C05457=1086.309,22.215,441.424,174.656,18.933,153.065
C05458=1086.315,22.464,441.409,174.658,18.935,153.065
C05459=1086.320,22.714,441.394,174.659,18.937,153.065
C05460=1086.326,22.963,441.379,174.661,18.939,153.065
C05461=1086.332,23.213,441.365,174.663,18.941,153.066
C05462=1086.337,23.462,441.350,174.664,18.942,153.066
C05463=1086.344,23.712,441.335,174.666,18.944,153.066
C05464=1086.349,23.961,441.320,174.667,18.946,153.066
C05465=1086.354,24.210,441.305,174.669,18.948,153.066
C05466=1086.361,24.460,441.290,174.671,18.951,153.066
C05467=1086.366,24.709,441.276,174.672,18.952,153.066
C05468=1086.372,24.959,441.261,174.674,18.954,153.066
C05469=1086.378,25.208,441.246,174.676,18.956,153.066
C05470=1086.384,25.458,441.231,174.677,18.958,153.066
C05471=1086.389,25.707,441.216,174.680,18.960,153.066
C05472=1086.395,25.957,441.201,174.681,18.962,153.066
C05473=1086.401,26.206,441.187,174.682,18.963,153.067
C05474=1086.407,26.456,441.171,174.684,18.966,153.067
C05475=1086.412,26.705,441.157,174.686,18.967,153.067
C05476=1086.419,26.955,441.142,174.687,18.969,153.067
C05477=1086.424,27.205,441.127,174.689,18.971,153.067
C05478=1086.430,27.454,441.112,174.691,18.973,153.067
C05479=1086.436,27.704,441.097,174.692,18.975,153.067
C05480=1086.442,27.953,441.082,174.694,18.977,153.067
C05481=1086.448,28.203,441.067,174.695,18.979,153.067
C05482=1086.453,28.452,441.052,174.697,18.980,153.067
C05483=1086.459,28.702,441.037,174.699,18.983,153.067
C05484=1086.464,28.951,441.022,174.700,18.984,153.067
C05485=1086.471,29.200,441.007,174.702,18.986,153.068
C05486=1086.476,29.450,440.992,174.704,18.988,153.068
C05487=1086.482,29.699,440.977,174.705,18.990,153.068
C05488=1086.487,29.949,440.962,174.706,18.992,153.068
C05489=1086.494,30.198,440.947,174.709,18.994,153.068
C05490=1086.499,30.448,440.931,174.710,18.996,153.068
C05491=1086.505,30.697,440.916,174.711,18.997,153.068
C05492=1086.512,30.975,440.899,174.713,19.000,153.068
C05493=1086.518,31.253,440.883,174.716,19.002,153.068
C05494=1086.524,31.531,440.866,174.717,19.004,153.068
C05495=1086.530,31.809,440.848,174.719,19.006,153.068
C05496=1086.536,32.058,440.833,174.720,19.008,153.069
C05497=1086.542,32.308,440.818,174.723,19.010,153.069
C05498=1086.548,32.557,440.803,174.724,19.012,153.069
C05499=1086.554,32.807,440.788,174.725,19.014,153.069
C05500=1086.559,33.056,440.773,174.728,19.016,153.069
C05501=1086.565,33.306,440.758,174.729,19.017,153.069
C05502=1086.571,33.555,440.743,174.731,19.020,153.069
C05503=1086.576,33.805,440.728,174.732,19.021,153.069
C05504=1086.582,34.055,440.712,174.734,19.023,153.069
C05505=1086.588,34.303,440.697,174.736,19.025,153.069
C05506=1086.594,34.553,440.681,174.737,19.027,153.069
C05507=1086.600,34.802,440.667,174.739,19.029,153.069
C05508=1086.605,35.052,440.651,174.741,19.031,153.069
C05509=1086.612,35.302,440.636,174.742,19.033,153.070
C05510=1086.617,35.551,440.620,174.745,19.035,153.070
C05511=1086.623,35.801,440.605,174.746,19.037,153.070
C05512=1086.629,36.050,440.590,174.747,19.038,153.070
C05513=1086.634,36.299,440.575,174.750,19.040,153.070
C05514=1086.640,36.549,440.560,174.751,19.042,153.070
C05515=1086.646,36.798,440.544,174.752,19.044,153.070
C05516=1086.651,37.048,440.528,174.754,19.046,153.070
C05517=1086.658,37.297,440.513,174.756,19.047,153.070
C05518=1086.663,37.547,440.498,174.758,19.050,153.070
C05519=1086.669,37.796,440.482,174.759,19.051,153.070
C05520=1086.675,38.046,440.467,174.761,19.053,153.070
C05521=1086.680,38.295,440.452,174.763,19.056,153.070
C05522=1086.686,38.545,440.436,174.764,19.057,153.070
C05523=1086.692,38.794,440.420,174.766,19.059,153.071
C05524=1086.698,39.043,440.405,174.768,19.061,153.071
C05525=1086.703,39.293,440.390,174.769,19.063,153.071
C05526=1086.709,39.543,440.373,174.772,19.065,153.071
C05527=1086.714,39.792,440.358,174.773,19.067,153.071
C05528=1086.721,40.041,440.343,174.774,19.068,153.071
C05529=1086.727,40.291,440.327,174.776,19.070,153.071
C05530=1086.732,40.540,440.312,174.778,19.072,153.071
C05531=1086.737,40.790,440.296,174.780,19.074,153.071
C05532=1086.744,41.039,440.281,174.781,19.076,153.071
C05533=1086.749,41.288,440.266,174.783,19.078,153.071
C05534=1086.755,41.538,440.250,174.785,19.080,153.071
C05535=1086.761,41.788,440.234,174.786,19.081,153.071
C05536=1086.766,42.037,440.219,174.788,19.084,153.072
C05537=1086.772,42.286,440.203,174.790,19.086,153.072
C05538=1086.778,42.536,440.187,174.791,19.087,153.072
C05539=1086.783,42.785,440.172,174.793,19.090,153.072
C05540=1086.789,43.035,440.156,174.795,19.091,153.072
C05541=1086.795,43.285,440.140,174.796,19.093,153.072
C05542=1086.801,43.534,440.124,174.798,19.095,153.072
C05543=1086.806,43.783,440.110,174.800,19.097,153.072
C05544=1086.812,44.032,440.093,174.802,19.099,153.072
C05545=1086.818,44.282,440.078,174.803,19.100,153.072
C05546=1086.823,44.531,440.062,174.805,19.102,153.072
C05547=1086.829,44.781,440.046,174.807,19.104,153.072
C05548=1086.835,45.030,440.030,174.808,19.106,153.072
C05549=1086.840,45.279,440.015,174.810,19.108,153.073
C05550=1086.846,45.529,439.999,174.812,19.110,153.073
C05551=1086.852,45.779,439.983,174.814,19.112,153.073
C05552=1086.857,46.027,439.967,174.815,19.114,153.073
C05553=1086.863,46.277,439.952,174.817,19.116,153.073
C05554=1086.868,46.527,439.935,174.819,19.118,153.073
C05555=1086.874,46.777,439.920,174.820,19.120,153.073
C05556=1086.880,47.055,439.902,174.822,19.122,153.073
C05557=1086.886,47.333,439.884,174.825,19.124,153.073
C05558=1086.893,47.610,439.867,174.826,19.126,153.073
C05559=1086.899,47.888,439.849,174.828,19.128,153.073
C05560=1086.904,48.138,439.833,174.829,19.130,153.073
C05561=1086.910,48.387,439.817,174.832,19.132,153.073
C05562=1086.916,48.636,439.801,174.833,19.134,153.074
C05563=1086.921,48.886,439.786,174.835,19.136,153.074
C05564=1086.927,49.135,439.769,174.837,19.137,153.074
C05565=1086.932,49.385,439.754,174.838,19.139,153.074
C05566=1086.938,49.634,439.738,174.840,19.141,153.074
C05567=1086.944,49.883,439.722,174.842,19.143,153.074
C05568=1086.950,50.133,439.706,174.844,19.145,153.074
C05569=1086.956,50.383,439.690,174.845,19.147,153.074
C05570=1086.961,50.631,439.674,174.847,19.149,153.074
C05571=1086.967,50.881,439.658,174.849,19.151,153.074
C05572=1086.972,51.131,439.642,174.850,19.152,153.074
C05573=1086.978,51.380,439.625,174.853,19.154,153.074
C05574=1086.984,51.630,439.610,174.854,19.156,153.074
C05575=1086.989,51.879,439.594,174.856,19.158,153.074
C05576=1086.995,52.128,439.578,174.857,19.160,153.074
C05577=1087.001,52.378,439.561,174.860,19.162,153.074
C05578=1087.007,52.628,439.546,174.861,19.164,153.075
C05579=1087.013,52.877,439.530,174.862,19.165,153.075
C05580=1087.018,53.126,439.514,174.865,19.167,153.075
C05581=1087.024,53.375,439.497,174.866,19.169,153.075
C05582=1087.029,53.625,439.482,174.868,19.171,153.075
C05583=1087.035,53.875,439.465,174.870,19.173,153.075
C05584=1087.041,54.124,439.449,174.872,19.175,153.075
C05585=1087.047,54.373,439.432,174.873,19.176,153.075
C05586=1087.053,54.623,439.416,174.875,19.178,153.075
C05587=1087.058,54.872,439.401,174.877,19.180,153.075
C05588=1087.064,55.121,439.385,174.878,19.182,153.075
C05589=1087.069,55.371,439.369,174.881,19.184,153.075
C05590=1087.075,55.620,439.352,174.882,19.186,153.075
C05591=1087.081,55.870,439.335,174.884,19.188,153.075
C05592=1087.087,56.119,439.319,174.886,19.189,153.075
C05593=1087.092,56.369,439.304,174.887,19.191,153.075
C05594=1087.098,56.618,439.287,174.890,19.193,153.075
C05595=1087.104,56.868,439.271,174.891,19.195,153.076
C05596=1087.110,57.117,439.255,174.893,19.197,153.076
C05597=1087.115,57.366,439.239,174.894,19.198,153.076
C05598=1087.121,57.615,439.222,174.897,19.200,153.076
C05599=1087.127,57.865,439.206,174.898,19.202,153.076
C05600=1087.133,58.114,439.190,174.901,19.204,153.076
C05601=1087.139,58.363,439.173,174.902,19.205,153.076
C05602=1087.144,58.613,439.157,174.903,19.207,153.076
C05603=1087.150,58.862,439.141,174.905,19.209,153.076
C05604=1087.155,59.112,439.125,174.907,19.211,153.076
C05605=1087.161,59.362,439.108,174.909,19.213,153.076
C05606=1087.167,59.611,439.092,174.911,19.215,153.076
C05607=1087.173,59.860,439.076,174.913,19.217,153.076
C05608=1087.179,60.110,439.060,174.914,19.218,153.076
C05609=1087.184,60.359,439.043,174.917,19.220,153.076
C05610=1087.190,60.609,439.027,174.918,19.222,153.076
C05611=1087.196,60.858,439.010,174.920,19.224,153.076
C05612=1087.202,61.107,438.994,174.922,19.225,153.076
C05613=1087.208,61.357,438.978,174.923,19.227,153.076
C05614=1087.214,61.606,438.960,174.926,19.229,153.076
C05615=1087.220,61.855,438.944,174.927,19.230,153.076
C05616=1087.226,62.104,438.928,174.929,19.233,153.076
C05617=1087.232,62.354,438.911,174.931,19.234,153.076
C05618=1087.237,62.603,438.895,174.933,19.236,153.076
C05619=1087.243,62.853,438.878,174.934,19.238,153.076
C05620=1087.249,63.130,438.860,174.937,19.240,153.076
C05621=1087.256,63.408,438.842,174.939,19.242,153.076
C05622=1087.262,63.686,438.824,174.940,19.243,153.077
C05623=1087.269,63.964,438.805,174.943,19.245,153.077
C05624=1087.275,64.213,438.789,174.945,19.247,153.077
C05625=1087.280,64.462,438.772,174.946,19.249,153.077
C05626=1087.286,64.712,438.755,174.948,19.251,153.077
C05627=1087.292,64.961,438.739,174.950,19.253,153.077
C05628=1087.297,65.211,438.722,174.952,19.254,153.077
C05629=1087.303,65.460,438.706,174.954,19.256,153.077
C05630=1087.308,65.710,438.689,174.955,19.258,153.077
C05631=1087.315,65.958,438.672,174.957,19.260,153.077
C05632=1087.320,66.208,438.655,174.959,19.262,153.077
C05633=1087.326,66.457,438.639,174.961,19.264,153.077
C05634=1087.332,66.707,438.623,174.963,19.265,153.077
C05635=1087.337,66.956,438.606,174.965,19.267,153.077
C05636=1087.344,67.206,438.589,174.966,19.269,153.077
C05637=1087.349,67.455,438.572,174.969,19.271,153.077
C05638=1087.355,67.705,438.556,174.970,19.272,153.077
C05639=1087.360,67.954,438.539,174.972,19.274,153.077
C05640=1087.366,68.203,438.522,174.974,19.276,153.077
C05641=1087.372,68.453,438.505,174.976,19.278,153.077
C05642=1087.378,68.702,438.489,174.978,19.279,153.077
C05643=1087.383,68.952,438.472,174.980,19.281,153.077
C05644=1087.389,69.201,438.455,174.981,19.283,153.077
C05645=1087.394,69.450,438.438,174.984,19.285,153.077
C05646=1087.400,69.700,438.422,174.985,19.286,153.077
C05647=1087.406,69.949,438.404,174.987,19.288,153.077
C05648=1087.412,70.198,438.388,174.989,19.290,153.077
C05649=1087.417,70.448,438.371,174.990,19.292,153.077
C05650=1087.422,70.697,438.353,174.992,19.294,153.077
C05651=1087.428,70.946,438.337,174.994,19.295,153.077
C05652=1087.434,71.196,438.320,174.996,19.297,153.077
C05653=1087.440,71.445,438.303,174.998,19.299,153.078
C05654=1087.446,71.695,438.286,175.000,19.301,153.078
C05655=1087.451,71.944,438.269,175.001,19.302,153.078
C05656=1087.457,72.193,438.252,175.004,19.304,153.078
C05657=1087.462,72.443,438.235,175.005,19.306,153.078
C05658=1087.469,72.691,438.218,175.007,19.308,153.078
C05659=1087.474,72.941,438.202,175.009,19.309,153.078
C05660=1087.479,73.191,438.185,175.011,19.311,153.078
C05661=1087.485,73.440,438.168,175.013,19.313,153.078
C05662=1087.490,73.689,438.151,175.015,19.315,153.078
C05663=1087.497,73.939,438.133,175.016,19.316,153.078
C05664=1087.503,74.188,438.117,175.019,19.318,153.078
C05665=1087.508,74.437,438.099,175.020,19.320,153.078
C05666=1087.513,74.687,438.082,175.022,19.322,153.078
C05667=1087.520,74.936,438.065,175.024,19.323,153.078
C05668=1087.525,75.185,438.049,175.026,19.325,153.078
C05669=1087.530,75.434,438.031,175.028,19.327,153.078
C05670=1087.537,75.684,438.014,175.030,19.329,153.078
C05671=1087.542,75.934,437.997,175.031,19.330,153.078
C05672=1087.548,76.183,437.980,175.034,19.332,153.078
C05673=1087.554,76.432,437.963,175.035,19.334,153.078
C05674=1087.559,76.682,437.946,175.038,19.336,153.078
C05675=1087.565,76.931,437.929,175.039,19.337,153.078
C05676=1087.571,77.180,437.911,175.041,19.339,153.078
C05677=1087.577,77.430,437.894,175.043,19.341,153.078
C05678=1087.582,77.679,437.877,175.045,19.343,153.078
C05679=1087.587,77.928,437.860,175.047,19.344,153.078
C05680=1087.593,78.177,437.842,175.049,19.346,153.078
C05681=1087.599,78.427,437.826,175.051,19.348,153.078
C05682=1087.605,78.677,437.808,175.053,19.350,153.078
C05683=1087.610,78.926,437.791,175.055,19.352,153.078
C05684=1087.617,79.203,437.772,175.056,19.353,153.078
C05685=1087.623,79.481,437.752,175.059,19.355,153.078
C05686=1087.629,79.758,437.734,175.061,19.357,153.078
C05687=1087.636,80.036,437.713,175.063,19.359,153.078
C05688=1087.641,80.286,437.697,175.065,19.361,153.078
C05689=1087.646,80.535,437.679,175.067,19.363,153.078
C05690=1087.652,80.784,437.661,175.069,19.364,153.078
C05691=1087.657,81.034,437.645,175.071,19.366,153.078
C05692=1087.664,81.283,437.627,175.073,19.367,153.078
C05693=1087.669,81.532,437.610,175.075,19.369,153.078
C05694=1087.675,81.782,437.593,175.076,19.371,153.078
C05695=1087.680,82.031,437.575,175.079,19.373,153.078
C05696=1087.689,82.421,437.547,175.082,19.375,153.078
C05697=1087.698,82.811,437.520,175.085,19.378,153.078
C05698=1087.707,83.200,437.494,175.088,19.381,153.078
C05699=1087.716,83.590,437.466,175.091,19.384,153.078
C05700=1087.721,83.839,437.449,175.092,19.385,153.078
C05701=1087.727,84.089,437.431,175.095,19.387,153.078
C05702=1087.733,84.338,437.413,175.096,19.389,153.078
C05703=1087.738,84.587,437.396,175.098,19.391,153.078
C05704=1087.744,84.836,437.378,175.100,19.392,153.078
C05705=1087.750,85.086,437.360,175.102,19.394,153.078
C05706=1087.755,85.336,437.344,175.105,19.396,153.078
C05707=1087.761,85.585,437.326,175.106,19.397,153.078
C05708=1087.767,85.835,437.308,175.108,19.399,153.078
C05709=1087.772,86.084,437.290,175.110,19.401,153.078
C05710=1087.778,86.333,437.273,175.112,19.402,153.078
C05711=1087.783,86.582,437.255,175.114,19.404,153.078
C05712=1087.789,86.831,437.237,175.116,19.406,153.078
C05713=1087.795,87.080,437.220,175.118,19.407,153.078
C05714=1087.800,87.329,437.202,175.120,19.409,153.078
C05715=1087.806,87.580,437.185,175.122,19.410,153.078
C05716=1087.812,87.829,437.168,175.124,19.412,153.078
C05717=1087.817,88.078,437.150,175.126,19.414,153.078
C05718=1087.823,88.328,437.132,175.128,19.415,153.078
C05719=1087.829,88.577,437.114,175.130,19.417,153.078
C05720=1087.834,88.826,437.097,175.132,19.419,153.078
C05721=1087.840,89.075,437.079,175.134,19.421,153.078
C05722=1087.846,89.325,437.061,175.136,19.422,153.078
C05723=1087.852,89.574,437.043,175.138,19.424,153.078
C05724=1087.858,89.823,437.026,175.139,19.425,153.078
C05725=1087.863,90.072,437.008,175.142,19.427,153.078
C05726=1087.869,90.322,436.990,175.144,19.429,153.078
C05727=1087.875,90.571,436.973,175.146,19.430,153.078
C05728=1087.880,90.820,436.955,175.148,19.432,153.078
C05729=1087.886,91.070,436.937,175.150,19.434,153.078
C05730=1087.892,91.319,436.920,175.152,19.436,153.078
C05731=1087.897,91.568,436.902,175.153,19.437,153.078
C05732=1087.903,91.817,436.883,175.156,19.439,153.078
C05733=1087.909,92.066,436.865,175.157,19.440,153.078
C05734=1087.915,92.316,436.847,175.160,19.442,153.078
C05735=1087.920,92.565,436.830,175.162,19.444,153.078
C05736=1087.925,92.815,436.812,175.164,19.445,153.078
C05737=1087.931,93.064,436.794,175.166,19.447,153.078
C05738=1087.937,93.313,436.776,175.168,19.449,153.078
C05739=1087.942,93.562,436.759,175.170,19.451,153.078
C05740=1087.948,93.812,436.741,175.172,19.452,153.078
C05741=1087.953,94.061,436.722,175.174,19.454,153.078
C05742=1087.959,94.310,436.704,175.176,19.456,153.078
C05743=1087.965,94.560,436.686,175.178,19.457,153.078
C05744=1087.974,94.947,436.658,175.181,19.459,153.078
C05745=1087.982,95.333,436.630,175.184,19.462,153.078
C05746=1087.991,95.720,436.602,175.187,19.465,153.078
C05747=1088.000,96.106,436.575,175.190,19.467,153.078
C05748=1088.006,96.355,436.556,175.193,19.469,153.078
C05749=1088.011,96.604,436.538,175.194,19.470,153.078
C05750=1088.017,96.854,436.520,175.197,19.472,153.078
C05751=1088.022,97.103,436.503,175.198,19.473,153.078
C05752=1088.028,97.353,436.483,175.200,19.475,153.078
C05753=1088.034,97.602,436.466,175.203,19.477,153.078
C05754=1088.040,97.851,436.448,175.204,19.478,153.078
C05755=1088.046,98.100,436.430,175.207,19.480,153.078
C05756=1088.051,98.350,436.411,175.208,19.481,153.078
C05757=1088.056,98.599,436.394,175.211,19.483,153.078
C05758=1088.063,98.849,436.376,175.213,19.485,153.078
C05759=1088.068,99.097,436.357,175.215,19.486,153.078
C05760=1088.073,99.346,436.339,175.217,19.488,153.077
C05761=1088.079,99.596,436.321,175.219,19.490,153.078
C05762=1088.085,99.846,436.302,175.221,19.492,153.078
C05763=1088.090,100.095,436.284,175.224,19.493,153.077
C05764=1088.097,100.344,436.266,175.225,19.495,153.077
C05765=1088.102,100.593,436.248,175.228,19.496,153.077
C05766=1088.108,100.843,436.230,175.229,19.498,153.077
C05767=1088.114,101.091,436.211,175.232,19.499,153.077
C05768=1088.119,101.341,436.193,175.234,19.501,153.077
C05769=1088.125,101.590,436.175,175.236,19.502,153.077
C05770=1088.130,101.840,436.156,175.238,19.504,153.077
C05771=1088.136,102.088,436.138,175.239,19.506,153.077
C05772=1088.141,102.338,436.119,175.242,19.507,153.077
C05773=1088.147,102.587,436.102,175.244,19.509,153.077
C05774=1088.153,102.837,436.082,175.246,19.510,153.077
C05775=1088.158,103.086,436.065,175.248,19.512,153.077
C05776=1088.164,103.335,436.046,175.250,19.513,153.077
C05777=1088.169,103.584,436.028,175.252,19.515,153.077
C05778=1088.175,103.834,436.009,175.255,19.517,153.077
C05779=1088.181,104.083,435.991,175.256,19.518,153.077
C05780=1088.186,104.332,435.972,175.259,19.520,153.077
C05781=1088.192,104.581,435.954,175.260,19.521,153.077
C05782=1088.197,104.831,435.935,175.263,19.523,153.077
C05783=1088.203,105.079,435.917,175.265,19.525,153.077
C05784=1088.209,105.329,435.898,175.267,19.526,153.077
C05785=1088.214,105.578,435.880,175.269,19.528,153.077
C05786=1088.220,105.828,435.862,175.271,19.530,153.077
C05787=1088.226,106.077,435.842,175.273,19.531,153.077
C05788=1088.231,106.326,435.825,175.275,19.533,153.077
C05789=1088.237,106.575,435.806,175.277,19.534,153.076
C05790=1088.243,106.824,435.787,175.279,19.536,153.076
C05791=1088.248,107.074,435.769,175.282,19.537,153.076
C05792=1088.253,107.323,435.750,175.283,19.539,153.076
C05793=1088.259,107.572,435.731,175.286,19.540,153.076
C05794=1088.265,107.822,435.713,175.287,19.542,153.076
C05795=1088.271,108.070,435.694,175.290,19.543,153.076
C05796=1088.276,108.320,435.676,175.292,19.545,153.076
C05797=1088.282,108.570,435.657,175.294,19.546,153.076
C05798=1088.288,108.818,435.638,175.296,19.548,153.076
C05799=1088.293,109.068,435.619,175.299,19.550,153.076
C05800=1088.299,109.317,435.602,175.300,19.551,153.076
C05801=1088.304,109.566,435.582,175.303,19.553,153.076
C05802=1088.310,109.816,435.563,175.305,19.555,153.076
C05803=1088.316,110.065,435.545,175.307,19.556,153.076
C05804=1088.321,110.314,435.526,175.309,19.558,153.076
C05805=1088.328,110.563,435.508,175.311,19.559,153.076
C05806=1088.333,110.812,435.489,175.314,19.560,153.075
C05807=1088.338,111.062,435.470,175.316,19.562,153.075
C05808=1088.345,111.339,435.449,175.318,19.564,153.075
C05809=1088.351,111.617,435.428,175.321,19.566,153.075
C05810=1088.358,111.895,435.407,175.323,19.567,153.075
C05811=1088.364,112.173,435.386,175.325,19.568,153.075
C05812=1088.369,112.422,435.367,175.327,19.570,153.075
C05813=1088.375,112.671,435.348,175.330,19.572,153.075
C05814=1088.381,112.921,435.330,175.331,19.573,153.075
C05815=1088.386,113.170,435.311,175.334,19.575,153.075
C05816=1088.392,113.419,435.292,175.336,19.576,153.075
C05817=1088.398,113.668,435.273,175.338,19.578,153.075
C05818=1088.403,113.917,435.254,175.340,19.579,153.075
C05819=1088.409,114.166,435.235,175.343,19.581,153.075
C05820=1088.414,114.416,435.216,175.344,19.582,153.075
C05821=1088.420,114.664,435.197,175.347,19.584,153.075
C05822=1088.426,114.914,435.179,175.349,19.586,153.075
C05823=1088.431,115.164,435.160,175.351,19.587,153.074
C05824=1088.436,115.412,435.141,175.353,19.588,153.074
C05825=1088.442,115.662,435.122,175.356,19.590,153.074
C05826=1088.448,115.911,435.102,175.357,19.591,153.074
C05827=1088.453,116.160,435.083,175.360,19.593,153.074
C05828=1088.459,116.409,435.064,175.362,19.595,153.074
C05829=1088.464,116.659,435.045,175.364,19.596,153.074
C05830=1088.469,116.908,435.026,175.366,19.598,153.074
C05831=1088.475,117.157,435.007,175.369,19.599,153.074
C05832=1088.481,117.406,434.988,175.371,19.600,153.074
C05833=1088.486,117.656,434.968,175.373,19.602,153.074
C05834=1088.491,117.905,434.949,175.375,19.604,153.074
C05835=1088.497,118.154,434.930,175.377,19.605,153.074
C05836=1088.503,118.403,434.911,175.379,19.607,153.074
C05837=1088.508,118.652,434.892,175.382,19.608,153.074
C05838=1088.514,118.902,434.873,175.384,19.609,153.073
C05839=1088.519,119.151,434.854,175.386,19.611,153.073
C05840=1088.525,119.400,434.834,175.388,19.613,153.073
C05841=1088.530,119.649,434.815,175.390,19.614,153.073
C05842=1088.536,119.898,434.796,175.392,19.616,153.073
C05843=1088.542,120.147,434.776,175.395,19.617,153.073
C05844=1088.547,120.397,434.757,175.397,19.618,153.073
C05845=1088.553,120.646,434.738,175.399,19.620,153.073
C05846=1088.558,120.895,434.719,175.402,19.622,153.073
C05847=1088.564,121.144,434.700,175.403,19.623,153.073
C05848=1088.570,121.394,434.680,175.406,19.625,153.073
C05849=1088.575,121.643,434.661,175.408,19.627,153.073
C05850=1088.581,121.891,434.642,175.410,19.628,153.073
C05851=1088.586,122.141,434.622,175.412,19.629,153.073
C05852=1088.592,122.390,434.603,175.415,19.631,153.072
C05853=1088.598,122.640,434.584,175.417,19.632,153.072
C05854=1088.603,122.889,434.565,175.419,19.634,153.072
C05855=1088.609,123.137,434.545,175.421,19.635,153.072
C05856=1088.615,123.387,434.526,175.424,19.637,153.072
C05857=1088.620,123.636,434.507,175.426,19.638,153.072
C05858=1088.626,123.886,434.487,175.428,19.639,153.072
C05859=1088.632,124.134,434.467,175.431,19.641,153.072
C05860=1088.638,124.384,434.448,175.432,19.642,153.072
C05861=1088.643,124.633,434.429,175.435,19.644,153.072
C05862=1088.648,124.882,434.410,175.437,19.645,153.072
C05863=1088.654,125.131,434.389,175.439,19.646,153.071
C05864=1088.659,125.381,434.370,175.442,19.648,153.071
C05865=1088.665,125.630,434.351,175.444,19.649,153.071
C05866=1088.671,125.879,434.331,175.446,19.651,153.071
C05867=1088.677,126.128,434.312,175.448,19.652,153.071
C05868=1088.682,126.378,434.292,175.451,19.654,153.071
C05869=1088.688,126.626,434.273,175.453,19.655,153.071
C05870=1088.693,126.875,434.254,175.455,19.656,153.071
C05871=1088.699,127.125,434.234,175.457,19.658,153.071
C05872=1088.706,127.402,434.212,175.460,19.659,153.071
C05873=1088.712,127.680,434.190,175.463,19.661,153.070
C05874=1088.718,127.958,434.169,175.465,19.662,153.070
C05875=1088.725,128.235,434.146,175.468,19.664,153.070
C05876=1088.730,128.485,434.127,175.470,19.666,153.070
C05877=1088.735,128.734,434.107,175.473,19.667,153.070
C05878=1088.741,128.983,434.087,175.474,19.668,153.070
C05879=1088.747,129.233,434.068,175.477,19.670,153.070
C05880=1088.753,129.481,434.048,175.479,19.671,153.070
C05881=1088.759,129.731,434.029,175.481,19.672,153.070
C05882=1088.765,129.980,434.009,175.484,19.674,153.069
C05883=1088.770,130.229,433.990,175.486,19.675,153.069
C05884=1088.776,130.478,433.969,175.489,19.677,153.069
C05885=1088.781,130.728,433.950,175.490,19.678,153.069
C05886=1088.787,130.976,433.930,175.493,19.679,153.069
C05887=1088.793,131.226,433.911,175.495,19.681,153.069
C05888=1088.799,131.475,433.891,175.498,19.682,153.069
C05889=1088.804,131.724,433.871,175.500,19.683,153.069
C05890=1088.810,131.973,433.851,175.502,19.685,153.069
C05891=1088.816,132.222,433.831,175.505,19.686,153.068
C05892=1088.822,132.471,433.812,175.506,19.687,153.068
C05893=1088.827,132.721,433.791,175.509,19.689,153.068
C05894=1088.833,132.970,433.772,175.512,19.691,153.068
C05895=1088.839,133.219,433.752,175.514,19.692,153.068
C05896=1088.844,133.468,433.732,175.516,19.693,153.068
C05897=1088.850,133.717,433.712,175.518,19.695,153.068
C05898=1088.855,133.967,433.692,175.521,19.696,153.068
C05899=1088.860,134.215,433.673,175.523,19.698,153.067
C05900=1088.866,134.464,433.653,175.525,19.699,153.067
C05901=1088.871,134.713,433.632,175.528,19.700,153.067
C05902=1088.877,134.963,433.613,175.530,19.702,153.067
C05903=1088.882,135.212,433.593,175.533,19.703,153.067
C05904=1088.888,135.461,433.573,175.534,19.704,153.067
C05905=1088.894,135.710,433.553,175.537,19.706,153.067
C05906=1088.900,135.960,433.532,175.540,19.707,153.067
C05907=1088.906,136.209,433.512,175.542,19.709,153.067
C05908=1088.911,136.458,433.492,175.544,19.710,153.066
C05909=1088.917,136.707,433.473,175.546,19.711,153.066
C05910=1088.923,136.956,433.453,175.549,19.713,153.066
C05911=1088.928,137.205,433.432,175.551,19.714,153.066
C05912=1088.934,137.454,433.412,175.553,19.715,153.066
C05913=1088.939,137.704,433.392,175.556,19.716,153.066
C05914=1088.945,137.953,433.372,175.558,19.718,153.066
C05915=1088.950,138.202,433.352,175.561,19.719,153.066
C05916=1088.956,138.450,433.332,175.563,19.720,153.065
C05917=1088.961,138.700,433.311,175.565,19.722,153.065
C05918=1088.967,138.949,433.292,175.568,19.723,153.065
C05919=1088.972,139.198,433.272,175.570,19.725,153.065
C05920=1088.978,139.447,433.252,175.572,19.726,153.065
C05921=1088.983,139.696,433.231,175.575,19.727,153.065
C05922=1088.989,139.945,433.211,175.577,19.729,153.065
C05923=1088.995,140.195,433.190,175.580,19.730,153.065
C05924=1089.001,140.444,433.170,175.582,19.731,153.064
C05925=1089.007,140.693,433.150,175.584,19.732,153.064
C05926=1089.012,140.942,433.130,175.587,19.734,153.064
C05927=1089.018,141.191,433.110,175.589,19.735,153.064
C05928=1089.023,141.440,433.089,175.592,19.737,153.064
C05929=1089.029,141.689,433.069,175.594,19.738,153.064
C05930=1089.034,141.938,433.049,175.596,19.739,153.064
C05931=1089.039,142.187,433.028,175.599,19.741,153.064
C05932=1089.045,142.436,433.008,175.601,19.742,153.063
C05933=1089.051,142.685,432.988,175.604,19.744,153.063
C05934=1089.056,142.935,432.967,175.606,19.744,153.063
C05935=1089.062,143.184,432.947,175.608,19.746,153.063
C05936=1089.068,143.461,432.924,175.611,19.747,153.063
C05937=1089.075,143.739,432.902,175.613,19.749,153.063
C05938=1089.081,144.017,432.878,175.616,19.750,153.063
C05939=1089.086,144.294,432.856,175.619,19.753,153.062
C05940=1089.093,144.544,432.835,175.621,19.753,153.062
C05941=1089.098,144.793,432.815,175.624,19.755,153.062
C05942=1089.104,145.042,432.794,175.626,19.756,153.062
C05943=1089.109,145.291,432.774,175.629,19.758,153.062
C05944=1089.115,145.540,432.754,175.631,19.759,153.062
C05945=1089.120,145.789,432.733,175.633,19.760,153.061
C05946=1089.126,146.039,432.712,175.636,19.761,153.061
C05947=1089.132,146.287,432.692,175.638,19.763,153.061
C05948=1089.137,146.536,432.671,175.641,19.764,153.061
C05949=1089.143,146.785,432.650,175.643,19.766,153.061
C05950=1089.149,147.034,432.630,175.645,19.766,153.061
C05951=1089.155,147.284,432.610,175.648,19.768,153.061
C05952=1089.160,147.533,432.589,175.650,19.769,153.061
C05953=1089.165,147.781,432.568,175.653,19.770,153.060
C05954=1089.171,148.030,432.548,175.656,19.772,153.060
C05955=1089.177,148.280,432.527,175.658,19.773,153.060
C05956=1089.182,148.529,432.506,175.660,19.774,153.060
C05957=1089.188,148.778,432.486,175.663,19.776,153.060
C05958=1089.194,149.027,432.465,175.665,19.777,153.060
C05959=1089.199,149.276,432.445,175.668,19.778,153.059
C05960=1089.205,149.526,432.424,175.670,19.779,153.059
C05961=1089.210,149.775,432.403,175.672,19.781,153.059
C05962=1089.216,150.023,432.382,175.675,19.782,153.059
C05963=1089.221,150.272,432.361,175.678,19.783,153.059
C05964=1089.227,150.522,432.340,175.680,19.785,153.059
C05965=1089.232,150.771,432.320,175.683,19.786,153.058
C05966=1089.239,151.019,432.299,175.685,19.787,153.058
C05967=1089.244,151.269,432.279,175.687,19.788,153.058
C05968=1089.249,151.518,432.258,175.690,19.790,153.058
C05969=1089.255,151.767,432.236,175.692,19.791,153.058
C05970=1089.261,152.016,432.216,175.695,19.792,153.058
C05971=1089.266,152.265,432.195,175.698,19.794,153.058
C05972=1089.272,152.514,432.174,175.699,19.795,153.058
C05973=1089.277,152.763,432.153,175.702,19.796,153.057
C05974=1089.283,153.012,432.132,175.705,19.797,153.057
C05975=1089.288,153.261,432.111,175.707,19.799,153.057
C05976=1089.294,153.511,432.090,175.710,19.800,153.057
C05977=1089.299,153.759,432.069,175.712,19.801,153.057
C05978=1089.305,154.009,432.048,175.714,19.803,153.057
C05979=1089.311,154.258,432.027,175.717,19.804,153.056
C05980=1089.316,154.507,432.006,175.719,19.805,153.056
C05981=1089.322,154.755,431.985,175.722,19.807,153.056
C05982=1089.328,155.005,431.965,175.725,19.808,153.056
C05983=1089.334,155.254,431.944,175.727,19.809,153.056
C05984=1089.339,155.502,431.923,175.729,19.810,153.055
C05985=1089.345,155.752,431.902,175.732,19.811,153.055
C05986=1089.350,156.001,431.880,175.734,19.813,153.055
C05987=1089.355,156.250,431.860,175.737,19.814,153.055
C05988=1089.361,156.499,431.838,175.740,19.815,153.055
C05989=1089.367,156.748,431.817,175.742,19.817,153.055
C05990=1089.372,156.997,431.796,175.745,19.818,153.054
C05991=1089.378,157.246,431.775,175.747,19.819,153.054
C05992=1089.383,157.495,431.754,175.749,19.820,153.054
C05993=1089.389,157.744,431.733,175.752,19.821,153.054
C05994=1089.395,157.994,431.712,175.755,19.823,153.054
C05995=1089.400,158.242,431.690,175.757,19.824,153.054
C05996=1089.406,158.491,431.669,175.760,19.825,153.053
C05997=1089.412,158.741,431.648,175.762,19.827,153.053
C05998=1089.417,158.989,431.626,175.765,19.828,153.053
C05999=1089.422,159.239,431.606,175.767,19.829,153.053
C06000=1089.428,159.516,431.582,175.771,19.830,153.053
C06001=1089.435,159.793,431.558,175.773,19.832,153.053
C06002=1089.441,160.071,431.534,175.776,19.833,153.052
C06003=1089.448,160.348,431.510,175.778,19.834,153.052
C06004=1089.453,160.597,431.490,175.781,19.835,153.052
C06005=1089.459,160.846,431.468,175.784,19.837,153.052
C06006=1089.465,161.095,431.447,175.787,19.838,153.052
C06007=1089.470,161.344,431.425,175.789,19.839,153.051
C06008=1089.475,161.593,431.404,175.792,19.840,153.051
C06009=1089.481,161.842,431.383,175.794,19.841,153.051
C06010=1089.487,162.091,431.361,175.796,19.843,153.051
C06011=1089.492,162.341,431.340,175.799,19.844,153.051
C06012=1089.497,162.589,431.319,175.801,19.846,153.051
C06013=1089.503,162.839,431.297,175.804,19.847,153.050
C06014=1089.508,163.087,431.275,175.807,19.848,153.050
C06015=1089.514,163.336,431.254,175.809,19.850,153.050
C06016=1089.519,163.586,431.233,175.812,19.851,153.050
C06017=1089.524,163.834,431.211,175.815,19.852,153.050
C06018=1089.530,164.084,431.189,175.817,19.854,153.050
C06019=1089.535,164.332,431.168,175.819,19.854,153.049
C06020=1089.541,164.581,431.146,175.822,19.856,153.049
C06021=1089.546,164.830,431.124,175.824,19.857,153.049
C06022=1089.552,165.079,431.103,175.827,19.858,153.049
C06023=1089.557,165.329,431.082,175.830,19.860,153.049
C06024=1089.563,165.577,431.060,175.832,19.861,153.049
C06025=1089.568,165.827,431.038,175.835,19.862,153.048
C06026=1089.574,166.075,431.017,175.837,19.864,153.048
C06027=1089.579,166.325,430.995,175.840,19.865,153.048
C06028=1089.585,166.573,430.973,175.843,19.866,153.048
C06029=1089.590,166.822,430.952,175.846,19.867,153.048
C06030=1089.595,167.071,430.930,175.847,19.868,153.048
C06031=1089.601,167.320,430.909,175.850,19.869,153.047
C06032=1089.606,167.570,430.886,175.853,19.871,153.047
C06033=1089.612,167.818,430.865,175.855,19.872,153.047
C06034=1089.617,168.068,430.843,175.858,19.873,153.047
C06035=1089.623,168.316,430.822,175.861,19.874,153.047
C06036=1089.628,168.566,430.799,175.863,19.876,153.046
C06037=1089.634,168.814,430.778,175.866,19.877,153.046
C06038=1089.639,169.064,430.756,175.869,19.878,153.046
C06039=1089.645,169.312,430.735,175.871,19.879,153.046
C06040=1089.650,169.562,430.712,175.874,19.881,153.046
C06041=1089.656,169.810,430.691,175.877,19.882,153.045
C06042=1089.661,170.060,430.669,175.879,19.884,153.045
C06043=1089.667,170.308,430.648,175.882,19.885,153.045
C06044=1089.672,170.558,430.625,175.884,19.886,153.045
C06045=1089.678,170.806,430.603,175.887,19.887,153.045
C06046=1089.684,171.055,430.581,175.889,19.888,153.044
C06047=1089.690,171.304,430.559,175.892,19.889,153.044
C06048=1089.695,171.553,430.538,175.895,19.890,153.044
C06049=1089.700,171.803,430.515,175.897,19.892,153.044
C06050=1089.706,172.051,430.494,175.900,19.893,153.044
C06051=1089.711,172.300,430.471,175.903,19.894,153.044
C06052=1089.717,172.548,430.450,175.905,19.895,153.043
C06053=1089.722,172.798,430.428,175.908,19.896,153.043
C06054=1089.729,173.047,430.406,175.911,19.898,153.043
C06055=1089.733,173.296,430.384,175.913,19.899,153.043
C06056=1089.739,173.545,430.361,175.916,19.900,153.043
C06057=1089.745,173.794,430.340,175.919,19.901,153.042
C06058=1089.750,174.043,430.318,175.922,19.902,153.042
C06059=1089.756,174.292,430.296,175.924,19.904,153.042
C06060=1089.761,174.540,430.273,175.927,19.905,153.042
C06061=1089.768,174.790,430.252,175.930,19.906,153.041
C06062=1089.773,175.039,430.230,175.932,19.907,153.041
C06063=1089.778,175.287,430.207,175.935,19.908,153.041
C06064=1089.785,175.565,430.183,175.938,19.909,153.041
C06065=1089.791,175.842,430.158,175.941,19.910,153.041
C06066=1089.797,176.118,430.133,175.943,19.912,153.040
C06067=1089.803,176.396,430.109,175.947,19.914,153.040
C06068=1089.809,176.645,430.087,175.949,19.915,153.040
C06069=1089.815,176.894,430.064,175.952,19.916,153.040
C06070=1089.820,177.143,430.043,175.955,19.917,153.040
C06071=1089.826,177.392,430.020,175.958,19.918,153.039
C06072=1089.832,177.641,429.998,175.960,19.919,153.039
C06073=1089.837,177.889,429.975,175.963,19.921,153.039
C06074=1089.843,178.138,429.954,175.966,19.922,153.039
C06075=1089.849,178.387,429.931,175.968,19.923,153.038
C06076=1089.854,178.637,429.909,175.971,19.924,153.038
C06077=1089.860,178.885,429.887,175.974,19.925,153.038
C06078=1089.865,179.134,429.864,175.976,19.926,153.038
C06079=1089.871,179.384,429.842,175.979,19.927,153.038
C06080=1089.877,179.632,429.820,175.981,19.928,153.037
C06081=1089.882,179.881,429.797,175.984,19.929,153.037
C06082=1089.888,180.130,429.775,175.987,19.930,153.037
C06083=1089.894,180.379,429.753,175.989,19.931,153.037
C06084=1089.900,180.628,429.730,175.992,19.932,153.036
C06085=1089.905,180.877,429.707,175.995,19.933,153.036
C06086=1089.911,181.126,429.686,175.998,19.934,153.036
C06087=1089.917,181.374,429.663,176.000,19.936,153.036
C06088=1089.922,181.624,429.641,176.003,19.937,153.036
C06089=1089.928,181.873,429.618,176.006,19.938,153.035
C06090=1089.934,182.121,429.596,176.009,19.939,153.035
C06091=1089.939,182.370,429.574,176.011,19.940,153.035
C06092=1089.945,182.619,429.551,176.014,19.941,153.034
C06093=1089.951,182.868,429.529,176.017,19.943,153.034
C06094=1089.957,183.117,429.506,176.020,19.944,153.034
C06095=1089.962,183.366,429.483,176.022,19.945,153.034
C06096=1089.968,183.615,429.460,176.025,19.946,153.034
C06097=1089.974,183.864,429.439,176.028,19.947,153.033
C06098=1089.979,184.112,429.416,176.031,19.948,153.033
C06099=1089.985,184.361,429.393,176.034,19.949,153.033
C06100=1089.991,184.611,429.371,176.037,19.950,153.033
C06101=1089.996,184.860,429.348,176.040,19.951,153.032
C06102=1090.003,185.108,429.326,176.042,19.953,153.032
C06103=1090.009,185.357,429.303,176.045,19.954,153.032
C06104=1090.013,185.606,429.280,176.048,19.955,153.032
C06105=1090.018,185.855,429.257,176.050,19.956,153.032
C06106=1090.024,186.104,429.234,176.053,19.957,153.031
C06107=1090.030,186.353,429.212,176.056,19.958,153.031
C06108=1090.035,186.602,429.190,176.059,19.960,153.031
C06109=1090.040,186.851,429.167,176.061,19.961,153.031
C06110=1090.046,187.100,429.144,176.064,19.962,153.030
C06111=1090.052,187.349,429.121,176.067,19.963,153.030
C06112=1090.058,187.597,429.098,176.069,19.965,153.030
C06113=1090.063,187.846,429.075,176.072,19.966,153.030
C06114=1090.067,188.096,429.052,176.075,19.967,153.030
C06115=1090.073,188.344,429.030,176.078,19.968,153.029
C06116=1090.079,188.593,429.007,176.080,19.969,153.029
C06117=1090.085,188.842,428.984,176.083,19.970,153.029
C06118=1090.090,189.091,428.961,176.086,19.971,153.029
C06119=1090.095,189.339,428.938,176.089,19.972,153.028
C06120=1090.101,189.588,428.915,176.091,19.974,153.028
C06121=1090.106,189.837,428.892,176.094,19.975,153.028
C06122=1090.112,190.086,428.869,176.097,19.976,153.028
C06123=1090.118,190.335,428.846,176.100,19.977,153.028
C06124=1090.123,190.584,428.823,176.103,19.978,153.027
C06125=1090.129,190.833,428.800,176.106,19.980,153.027
C06126=1090.134,191.081,428.777,176.109,19.981,153.027
C06127=1090.139,191.330,428.754,176.111,19.982,153.027
C06128=1090.145,191.607,428.729,176.114,19.983,153.026
C06129=1090.152,191.884,428.703,176.118,19.985,153.026
C06130=1090.158,192.161,428.678,176.121,19.986,153.026
C06131=1090.164,192.438,428.651,176.123,19.987,153.026
C06132=1090.170,192.686,428.629,176.127,19.988,153.025
C06133=1090.175,192.935,428.606,176.129,19.990,153.025
C06134=1090.180,193.184,428.582,176.132,19.991,153.025
C06135=1090.186,193.433,428.559,176.135,19.992,153.025
C06136=1090.192,193.682,428.536,176.138,19.993,153.024
C06137=1090.198,193.930,428.513,176.141,19.994,153.024
C06138=1090.203,194.180,428.489,176.143,19.995,153.024
C06139=1090.209,194.428,428.466,176.146,19.996,153.024
C06140=1090.214,194.677,428.443,176.149,19.997,153.024
C06141=1090.220,194.926,428.420,176.152,19.998,153.023
C06142=1090.225,195.175,428.397,176.154,19.999,153.023
C06143=1090.231,195.424,428.373,176.157,20.001,153.023
C06144=1090.237,195.673,428.350,176.161,20.002,153.023
C06145=1090.242,195.922,428.327,176.163,20.003,153.022
C06146=1090.247,196.171,428.304,176.166,20.004,153.022
C06147=1090.253,196.420,428.281,176.169,20.005,153.022
C06148=1090.259,196.668,428.257,176.172,20.006,153.022
C06149=1090.265,196.917,428.234,176.175,20.007,153.021
C06150=1090.270,197.166,428.211,176.177,20.008,153.021
C06151=1090.276,197.415,428.188,176.180,20.009,153.021
C06152=1090.282,197.663,428.164,176.183,20.011,153.021
C06153=1090.287,197.912,428.140,176.186,20.012,153.020
C06154=1090.292,198.161,428.118,176.189,20.013,153.020
C06155=1090.298,198.410,428.094,176.192,20.014,153.020
C06156=1090.304,198.659,428.070,176.195,20.015,153.020
C06157=1090.310,198.908,428.047,176.197,20.016,153.019
C06158=1090.316,199.157,428.023,176.200,20.017,153.019
C06159=1090.321,199.406,428.000,176.203,20.019,153.019
C06160=1090.327,199.654,427.976,176.206,20.020,153.019
C06161=1090.333,199.903,427.953,176.209,20.021,153.018
C06162=1090.338,200.152,427.930,176.212,20.022,153.018
C06163=1090.344,200.401,427.906,176.215,20.023,153.018
C06164=1090.349,200.649,427.883,176.218,20.024,153.018
C06165=1090.355,200.898,427.859,176.221,20.025,153.017
C06166=1090.361,201.148,427.835,176.223,20.026,153.017
C06167=1090.367,201.396,427.812,176.226,20.027,153.017
C06168=1090.372,201.645,427.788,176.229,20.028,153.017
C06169=1090.378,201.893,427.765,176.232,20.029,153.016
C06170=1090.383,202.143,427.741,176.235,20.031,153.016
C06171=1090.389,202.391,427.717,176.238,20.032,153.016
C06172=1090.395,202.640,427.694,176.241,20.033,153.016
C06173=1090.401,202.889,427.670,176.244,20.034,153.015
C06174=1090.406,203.138,427.647,176.246,20.035,153.015
C06175=1090.412,203.387,427.623,176.249,20.036,153.015
C06176=1090.417,203.636,427.599,176.253,20.038,153.015
C06177=1090.423,203.884,427.575,176.256,20.039,153.014
C06178=1090.428,204.133,427.552,176.258,20.040,153.014
C06179=1090.434,204.381,427.528,176.261,20.041,153.014
C06180=1090.440,204.631,427.504,176.264,20.042,153.014
C06181=1090.445,204.880,427.480,176.267,20.043,153.013
C06182=1090.451,205.128,427.456,176.269,20.044,153.013
C06183=1090.456,205.377,427.433,176.273,20.045,153.013
C06184=1090.462,205.626,427.409,176.276,20.046,153.013
C06185=1090.467,205.874,427.385,176.279,20.047,153.012
C06186=1090.472,206.124,427.361,176.281,20.048,153.012
C06187=1090.479,206.373,427.337,176.284,20.050,153.012
C06188=1090.484,206.621,427.313,176.287,20.051,153.012
C06189=1090.489,206.870,427.289,176.291,20.052,153.011
C06190=1090.495,207.119,427.266,176.293,20.053,153.011
C06191=1090.500,207.367,427.242,176.296,20.054,153.011
C06192=1090.524,208.388,427.143,176.362,20.087,153.007
C06193=1090.532,208.770,427.106,176.367,20.090,153.007
C06194=1090.541,209.149,427.069,176.371,20.093,153.006
C06195=1090.550,209.529,427.032,176.375,20.096,153.006
C06196=1090.558,209.909,426.994,176.380,20.099,153.006
C06197=1090.564,210.158,426.970,176.383,20.101,153.006
C06198=1090.569,210.406,426.945,176.385,20.103,153.006
C06199=1090.574,210.655,426.921,176.388,20.106,153.006
C06200=1090.581,210.904,426.897,176.391,20.108,153.006
C06201=1090.586,211.153,426.873,176.394,20.110,153.006
C06202=1090.592,211.402,426.848,176.397,20.112,153.006
C06203=1090.598,211.650,426.823,176.400,20.114,153.006
C06204=1090.603,211.898,426.799,176.402,20.116,153.006
C06205=1090.609,212.148,426.774,176.405,20.118,153.006
C06206=1090.614,212.396,426.750,176.408,20.120,153.006
C06207=1090.620,212.646,426.726,176.411,20.122,153.006
C06208=1090.626,212.894,426.701,176.414,20.124,153.006
C06209=1090.631,213.142,426.676,176.416,20.126,153.006
C06210=1090.637,213.391,426.652,176.419,20.128,153.006
C06211=1090.642,213.640,426.627,176.422,20.130,153.006
C06212=1090.649,213.889,426.602,176.425,20.132,153.006
C06213=1090.653,214.138,426.577,176.427,20.134,153.006
C06214=1090.658,214.386,426.553,176.431,20.136,153.006
C06215=1090.664,214.635,426.528,176.433,20.138,153.006
C06216=1090.670,214.883,426.503,176.436,20.140,153.006
C06217=1090.676,215.133,426.479,176.439,20.142,153.006
C06218=1090.681,215.381,426.455,176.442,20.145,153.006
C06219=1090.687,215.630,426.429,176.444,20.146,153.006
C06220=1090.693,215.879,426.405,176.448,20.149,153.006
C06221=1090.697,216.127,426.380,176.450,20.151,153.006
C06222=1090.703,216.376,426.355,176.453,20.153,153.005
C06223=1090.709,216.625,426.330,176.456,20.155,153.006
C06224=1090.715,216.873,426.305,176.459,20.157,153.005
C06225=1090.720,217.122,426.281,176.461,20.159,153.005
C06226=1090.726,217.371,426.256,176.464,20.161,153.005
C06227=1090.731,217.620,426.231,176.467,20.163,153.005
C06228=1090.737,217.869,426.206,176.470,20.165,153.005
C06229=1090.742,218.117,426.181,176.473,20.167,153.005
C06230=1090.748,218.366,426.156,176.476,20.169,153.005
C06231=1090.754,218.614,426.132,176.478,20.171,153.005
C06232=1090.760,218.863,426.107,176.482,20.173,153.005
C06233=1090.765,219.112,426.081,176.484,20.175,153.005
C06234=1090.771,219.360,426.056,176.487,20.177,153.005
C06235=1090.777,219.610,426.031,176.490,20.179,153.005
C06236=1090.782,219.858,426.006,176.493,20.182,153.005
C06237=1090.788,220.107,425.981,176.495,20.183,153.005
C06238=1090.793,220.355,425.956,176.499,20.186,153.005
C06239=1090.799,220.604,425.932,176.501,20.188,153.005
C06240=1090.805,220.853,425.906,176.504,20.190,153.005
C06241=1090.811,221.101,425.881,176.507,20.192,153.005
C06242=1090.816,221.351,425.856,176.510,20.194,153.005
C06243=1090.822,221.599,425.831,176.512,20.196,153.005
C06244=1090.828,221.847,425.806,176.516,20.198,153.005
C06245=1090.837,222.232,425.767,176.520,20.201,153.005
C06246=1090.845,222.615,425.728,176.525,20.205,153.005
C06247=1090.853,222.999,425.690,176.529,20.208,153.005
C06248=1090.862,223.383,425.650,176.534,20.211,153.005
C06249=1090.867,223.632,425.625,176.536,20.213,153.005
C06250=1090.873,223.880,425.599,176.539,20.216,153.005
C06251=1090.878,224.129,425.574,176.542,20.217,153.005
C06252=1090.884,224.378,425.549,176.545,20.220,153.005
C06253=1090.890,224.627,425.524,176.547,20.222,153.005
C06254=1090.895,224.875,425.498,176.550,20.224,153.005
C06255=1090.902,225.123,425.473,176.553,20.226,153.005
C06256=1090.907,225.373,425.448,176.556,20.228,153.004
C06257=1090.912,225.621,425.423,176.559,20.230,153.004
C06258=1090.918,225.870,425.397,176.562,20.232,153.004
C06259=1090.924,226.119,425.371,176.565,20.234,153.004
C06260=1090.929,226.367,425.346,176.567,20.236,153.004
C06261=1090.935,226.616,425.321,176.571,20.239,153.004
C06262=1090.940,226.865,425.295,176.573,20.240,153.004
C06263=1090.946,227.113,425.270,176.576,20.243,153.004
C06264=1090.952,227.362,425.244,176.579,20.245,153.004
C06265=1090.958,227.610,425.218,176.582,20.247,153.004
C06266=1090.963,227.859,425.193,176.584,20.249,153.004
C06267=1090.969,228.108,425.168,176.588,20.251,153.004
C06268=1090.974,228.357,425.142,176.591,20.253,153.004
C06269=1090.980,228.605,425.117,176.593,20.255,153.004
C06270=1090.985,228.854,425.091,176.597,20.257,153.004
C06271=1090.992,229.102,425.065,176.599,20.259,153.004
C06272=1090.997,229.351,425.039,176.602,20.261,153.004
C06273=1091.003,229.600,425.013,176.605,20.263,153.004
C06274=1091.008,229.848,424.988,176.608,20.266,153.004
C06275=1091.014,230.097,424.963,176.611,20.268,153.004
C06276=1091.020,230.345,424.937,176.614,20.270,153.004
C06277=1091.025,230.594,424.911,176.617,20.272,153.004
C06278=1091.030,230.843,424.886,176.619,20.274,153.004
C06279=1091.036,231.091,424.860,176.623,20.276,153.004
C06280=1091.042,231.340,424.834,176.625,20.278,153.004
C06281=1091.048,231.589,424.808,176.628,20.280,153.004
C06282=1091.053,231.837,424.783,176.631,20.283,153.004
C06283=1091.059,232.086,424.757,176.634,20.285,153.004
C06284=1091.064,232.335,424.731,176.637,20.287,153.004
C06285=1091.070,232.584,424.705,176.639,20.289,153.004
C06286=1091.076,232.832,424.680,176.643,20.291,153.004
C06287=1091.081,233.080,424.653,176.646,20.294,153.004
C06288=1091.086,233.329,424.627,176.648,20.295,153.004
C06289=1091.092,233.578,424.602,176.652,20.298,153.004
C06290=1091.098,233.827,424.576,176.654,20.300,153.004
C06291=1091.104,234.075,424.550,176.657,20.302,153.004
C06292=1091.109,234.323,424.524,176.660,20.305,153.004
C06293=1091.114,234.572,424.498,176.663,20.307,153.004
C06294=1091.120,234.820,424.471,176.666,20.309,153.004
C06295=1091.126,235.069,424.446,176.669,20.311,153.004
C06296=1091.132,235.318,424.420,176.672,20.313,153.004
C06297=1091.140,235.693,424.380,176.677,20.317,153.004
C06298=1091.148,236.068,424.341,176.681,20.320,153.004
C06299=1091.157,236.444,424.302,176.685,20.323,153.004
C06300=1091.165,236.819,424.262,176.690,20.326,153.004
C06301=1091.171,237.068,424.236,176.693,20.329,153.004
C06302=1091.176,237.316,424.210,176.695,20.330,153.004
C06303=1091.182,237.565,424.183,176.698,20.333,153.004
C06304=1091.187,237.814,424.157,176.701,20.335,153.004
C06305=1091.193,238.062,424.131,176.704,20.337,153.004
C06306=1091.199,238.311,424.106,176.707,20.339,153.003
C06307=1091.205,238.559,424.079,176.710,20.341,153.004
C06308=1091.210,238.807,424.053,176.713,20.344,153.004
C06309=1091.216,239.056,424.027,176.716,20.346,153.003
C06310=1091.221,239.305,424.001,176.719,20.348,153.003
C06311=1091.227,239.553,423.974,176.722,20.350,153.003
C06312=1091.233,239.802,423.947,176.724,20.352,153.003
C06313=1091.238,240.051,423.921,176.728,20.354,153.003
C06314=1091.244,240.299,423.895,176.731,20.357,153.003
C06315=1091.250,240.548,423.869,176.733,20.359,153.003
C06316=1091.255,240.796,423.842,176.736,20.361,153.003
C06317=1091.261,241.045,423.816,176.740,20.363,153.003
C06318=1091.267,241.294,423.790,176.742,20.365,153.003
C06319=1091.272,241.542,423.763,176.745,20.367,153.003
C06320=1091.278,241.790,423.736,176.749,20.370,153.003
C06321=1091.284,242.039,423.710,176.751,20.372,153.003
C06322=1091.289,242.288,423.684,176.754,20.374,153.003
C06323=1091.295,242.536,423.657,176.757,20.376,153.003
C06324=1091.301,242.784,423.631,176.760,20.378,153.003
C06325=1091.306,243.033,423.605,176.763,20.381,153.003
C06326=1091.312,243.282,423.578,176.766,20.383,153.003
C06327=1091.317,243.530,423.551,176.769,20.385,153.003
C06328=1091.323,243.779,423.524,176.772,20.387,153.003
C06329=1091.329,244.027,423.497,176.775,20.390,153.003
C06330=1091.334,244.276,423.471,176.777,20.392,153.003
C06331=1091.340,244.524,423.445,176.781,20.394,153.003
C06332=1091.345,244.773,423.418,176.784,20.396,153.003
C06333=1091.351,245.021,423.391,176.786,20.398,153.003
C06334=1091.357,245.270,423.364,176.789,20.401,153.003
C06335=1091.362,245.518,423.338,176.793,20.403,153.003
C06336=1091.368,245.767,423.311,176.795,20.405,153.003
C06337=1091.373,246.016,423.284,176.798,20.407,153.003
C06338=1091.379,246.264,423.258,176.802,20.410,153.003
C06339=1091.384,246.513,423.231,176.804,20.412,153.003
C06340=1091.390,246.761,423.204,176.807,20.414,153.003
C06341=1091.395,247.010,423.177,176.810,20.416,153.003
C06342=1091.402,247.259,423.150,176.813,20.418,153.003
C06343=1091.407,247.507,423.124,176.816,20.421,153.003
C06344=1091.412,247.756,423.096,176.819,20.423,153.003
C06345=1091.418,248.004,423.070,176.822,20.426,153.003
C06346=1091.424,248.252,423.043,176.825,20.428,153.003
C06347=1091.429,248.501,423.016,176.828,20.430,153.003
C06348=1091.435,248.749,422.989,176.831,20.432,153.003
C06349=1091.443,249.118,422.949,176.835,20.436,153.003
C06350=1091.451,249.486,422.909,176.840,20.439,153.003
C06351=1091.459,249.854,422.869,176.844,20.442,153.003
C06352=1091.468,250.223,422.829,176.849,20.446,153.004
C06353=1091.473,250.471,422.802,176.851,20.448,153.004
C06354=1091.479,250.719,422.775,176.854,20.450,153.003
C06355=1091.484,250.968,422.747,176.858,20.453,153.003
C06356=1091.490,251.216,422.721,176.860,20.455,153.004
C06357=1091.495,251.466,422.693,176.863,20.457,153.004
C06358=1091.501,251.714,422.667,176.866,20.460,153.004
C06359=1091.506,251.962,422.639,176.869,20.462,153.004
C06360=1091.512,252.210,422.612,176.872,20.464,153.004
C06361=1091.517,252.459,422.585,176.875,20.467,153.004
C06362=1091.523,252.707,422.558,176.878,20.469,153.004
C06363=1091.529,252.956,422.530,176.882,20.471,153.004
C06364=1091.535,253.205,422.503,176.884,20.473,153.004
C06365=1091.540,253.453,422.476,176.887,20.476,153.004
C06366=1091.546,253.701,422.448,176.890,20.478,153.004
C06367=1091.551,253.950,422.421,176.893,20.480,153.004
C06368=1091.557,254.199,422.394,176.896,20.483,153.004
C06369=1091.562,254.447,422.366,176.899,20.485,153.004
C06370=1091.568,254.695,422.340,176.902,20.488,153.004
C06371=1091.573,254.944,422.312,176.905,20.489,153.004
C06372=1091.579,255.192,422.284,176.908,20.492,153.004
C06373=1091.585,255.441,422.257,176.911,20.494,153.004
C06374=1091.590,255.689,422.229,176.914,20.497,153.004
C06375=1091.596,255.937,422.203,176.917,20.499,153.004
C06376=1091.601,256.186,422.175,176.920,20.501,153.004
C06377=1091.608,256.434,422.148,176.923,20.504,153.004
C06378=1091.613,256.683,422.121,176.926,20.506,153.004
C06379=1091.618,256.931,422.093,176.929,20.508,153.004
C06380=1091.625,257.180,422.066,176.932,20.510,153.004
C06381=1091.630,257.428,422.038,176.935,20.513,153.004
C06382=1091.636,257.677,422.011,176.938,20.515,153.004
C06383=1091.641,257.925,421.983,176.941,20.517,153.004
C06384=1091.647,258.173,421.955,176.944,20.520,153.004
C06385=1091.653,258.422,421.928,176.947,20.522,153.004
C06386=1091.658,258.670,421.900,176.950,20.524,153.004
C06387=1091.664,258.919,421.873,176.953,20.526,153.004
C06388=1091.670,259.167,421.845,176.956,20.529,153.004
C06389=1091.676,259.416,421.817,176.959,20.531,153.004
C06390=1091.682,259.664,421.790,176.962,20.534,153.004
C06391=1091.687,259.912,421.762,176.965,20.536,153.004
C06392=1091.693,260.161,421.734,176.968,20.538,153.004
C06393=1091.699,260.409,421.707,176.971,20.540,153.004
C06394=1091.704,260.657,421.679,176.974,20.543,153.004
C06395=1091.710,260.906,421.651,176.978,20.545,153.004
C06396=1091.716,261.154,421.624,176.980,20.547,153.004
C06397=1091.722,261.403,421.596,176.983,20.550,153.004
C06398=1091.727,261.651,421.568,176.986,20.552,153.004
C06399=1091.733,261.899,421.541,176.990,20.555,153.004
C06400=1091.739,262.148,421.513,176.992,20.557,153.004
C06401=1091.747,262.513,421.472,176.997,20.560,153.004
C06402=1091.756,262.878,421.431,177.002,20.564,153.004
C06403=1091.763,263.244,421.390,177.006,20.567,153.004
C06404=1091.773,263.610,421.349,177.010,20.571,153.004
C06405=1091.778,263.858,421.321,177.014,20.573,153.004
C06406=1091.784,264.107,421.292,177.016,20.575,153.004
C06407=1091.790,264.354,421.265,177.019,20.577,153.004
C06408=1091.796,264.604,421.237,177.022,20.580,153.004
C06409=1091.801,264.852,421.209,177.026,20.582,153.004
C06410=1091.806,265.100,421.181,177.029,20.585,153.004
C06411=1091.812,265.349,421.153,177.031,20.586,153.004
C06412=1091.818,265.597,421.125,177.034,20.589,153.004
C06413=1091.824,265.845,421.097,177.038,20.591,153.005
C06414=1091.829,266.093,421.069,177.041,20.594,153.005
C06415=1091.835,266.342,421.041,177.044,20.596,153.005
C06416=1091.840,266.590,421.013,177.046,20.598,153.005
C06417=1091.846,266.839,420.984,177.050,20.601,153.005
C06418=1091.852,267.087,420.956,177.052,20.604,153.005
C06419=1091.858,267.336,420.928,177.056,20.606,153.005
C06420=1091.863,267.583,420.899,177.059,20.609,153.005
C06421=1091.869,267.831,420.871,177.061,20.611,153.005
C06422=1091.874,268.080,420.843,177.064,20.613,153.005
C06423=1091.880,268.328,420.815,177.068,20.616,153.005
C06424=1091.886,268.577,420.787,177.071,20.618,153.005
C06425=1091.892,268.826,420.758,177.074,20.621,153.005
C06426=1091.897,269.074,420.730,177.077,20.623,153.005
C06427=1091.903,269.322,420.702,177.079,20.625,153.005
C06428=1091.909,269.570,420.673,177.083,20.628,153.005
C06429=1091.915,269.819,420.645,177.086,20.630,153.005
C06430=1091.920,270.067,420.617,177.089,20.633,153.005
C06431=1091.925,270.316,420.588,177.092,20.635,153.005
C06432=1091.931,270.563,420.560,177.095,20.638,153.005
C06433=1091.937,270.812,420.531,177.098,20.640,153.005
C06434=1091.942,271.060,420.503,177.101,20.642,153.005
C06435=1091.948,271.309,420.475,177.104,20.645,153.006
C06436=1091.954,271.556,420.446,177.107,20.648,153.006
C06437=1091.960,271.805,420.418,177.110,20.650,153.006
C06438=1091.965,272.054,420.389,177.114,20.653,153.006
C06439=1091.970,272.301,420.360,177.117,20.655,153.006
C06440=1091.976,272.550,420.332,177.119,20.657,153.006
C06441=1091.982,272.798,420.304,177.122,20.660,153.006
C06442=1091.988,273.046,420.275,177.125,20.662,153.006
C06443=1091.993,273.295,420.246,177.128,20.665,153.006
C06444=1091.999,273.543,420.217,177.132,20.668,153.006
C06445=1092.005,273.791,420.189,177.135,20.670,153.006
C06446=1092.010,274.039,420.160,177.138,20.672,153.006
C06447=1092.016,274.288,420.132,177.140,20.674,153.006
C06448=1092.022,274.537,420.103,177.144,20.677,153.006
C06449=1092.027,274.784,420.075,177.147,20.680,153.006
C06450=1092.032,275.033,420.046,177.150,20.682,153.006
C06451=1092.038,275.281,420.017,177.153,20.685,153.006
C06452=1092.044,275.529,419.989,177.156,20.687,153.007
C06453=1092.052,275.897,419.945,177.161,20.691,153.007
C06454=1092.061,276.266,419.902,177.165,20.695,153.007
C06455=1092.069,276.634,419.860,177.170,20.698,153.007
C06456=1092.078,277.002,419.817,177.174,20.702,153.007
C06457=1092.083,277.251,419.788,177.177,20.705,153.007
C06458=1092.089,277.499,419.759,177.180,20.708,153.007
C06459=1092.095,277.746,419.731,177.183,20.710,153.007
C06460=1092.100,277.996,419.702,177.186,20.712,153.007
C06461=1092.106,278.244,419.673,177.189,20.715,153.007
C06462=1092.111,278.491,419.643,177.192,20.718,153.007
C06463=1092.117,278.740,419.615,177.195,20.720,153.007
C06464=1092.123,278.988,419.586,177.198,20.723,153.007
C06465=1092.128,279.236,419.557,177.202,20.725,153.008
C06466=1092.134,279.484,419.528,177.205,20.728,153.008
C06467=1092.140,279.733,419.499,177.208,20.730,153.008
C06468=1092.146,279.981,419.470,177.211,20.733,153.008
C06469=1092.151,280.229,419.440,177.213,20.735,153.008
C06470=1092.157,280.477,419.411,177.216,20.738,153.008
C06471=1092.163,280.726,419.382,177.220,20.740,153.008
C06472=1092.169,280.974,419.353,177.223,20.743,153.008
C06473=1092.173,281.222,419.324,177.226,20.746,153.008
C06474=1092.180,281.470,419.295,177.229,20.748,153.008
C06475=1092.185,281.719,419.266,177.232,20.751,153.008
C06476=1092.191,281.967,419.236,177.235,20.754,153.008
C06477=1092.196,282.215,419.207,177.238,20.756,153.009
C06478=1092.202,282.463,419.178,177.241,20.759,153.009
C06479=1092.208,282.711,419.149,177.244,20.762,153.009
C06480=1092.214,282.960,419.119,177.248,20.764,153.009
C06481=1092.219,283.207,419.090,177.251,20.767,153.009
C06482=1092.225,283.455,419.061,177.253,20.769,153.009
C06483=1092.230,283.704,419.031,177.256,20.772,153.009
C06484=1092.236,283.952,419.001,177.259,20.774,153.009
C06485=1092.242,284.201,418.972,177.262,20.777,153.009
C06486=1092.247,284.448,418.943,177.265,20.780,153.009
C06487=1092.252,284.697,418.913,177.269,20.782,153.010
C06488=1092.259,284.945,418.884,177.272,20.785,153.010
C06489=1092.264,285.193,418.855,177.275,20.788,153.010
C06490=1092.270,285.442,418.825,177.278,20.790,153.010
C06491=1092.276,285.690,418.796,177.281,20.793,153.010
C06492=1092.281,285.938,418.767,177.284,20.796,153.010
C06493=1092.286,286.186,418.737,177.287,20.798,153.010
C06494=1092.292,286.434,418.707,177.290,20.801,153.010
C06495=1092.299,286.682,418.678,177.293,20.804,153.010
C06496=1092.304,286.930,418.648,177.296,20.807,153.010
C06497=1092.310,287.179,418.618,177.300,20.809,153.010
C06498=1092.315,287.427,418.589,177.303,20.812,153.011
C06499=1092.321,287.674,418.559,177.306,20.815,153.011
C06500=1092.327,287.923,418.530,177.309,20.817,153.011
C06501=1092.332,288.171,418.500,177.311,20.819,153.011
C06502=1092.338,288.419,418.471,177.314,20.822,153.011
C06503=1092.344,288.667,418.441,177.317,20.825,153.011
C06504=1092.350,288.915,418.411,177.321,20.827,153.011
C06505=1092.358,289.293,418.366,177.325,20.831,153.011
C06506=1092.367,289.671,418.321,177.330,20.836,153.012
C06507=1092.376,290.049,418.276,177.335,20.840,153.012
C06508=1092.384,290.426,418.230,177.340,20.844,153.012
C06509=1092.390,290.674,418.200,177.343,20.847,153.012
C06510=1092.395,290.922,418.170,177.346,20.850,153.012
C06511=1092.401,291.171,418.141,177.349,20.852,153.012
C06512=1092.407,291.418,418.111,177.352,20.855,153.012
C06513=1092.412,291.667,418.081,177.355,20.858,153.012
C06514=1092.418,291.915,418.051,177.358,20.861,153.013
C06515=1092.423,292.163,418.021,177.362,20.863,153.013
C06516=1092.429,292.411,417.991,177.365,20.866,153.013
C06517=1092.435,292.659,417.961,177.368,20.869,153.013
C06518=1092.441,292.907,417.931,177.371,20.872,153.013
C06519=1092.446,293.156,417.901,177.374,20.875,153.013
C06520=1092.452,293.404,417.871,177.377,20.877,153.013
C06521=1092.458,293.651,417.840,177.380,20.880,153.013
C06522=1092.463,293.900,417.811,177.383,20.883,153.014
C06523=1092.469,294.148,417.780,177.386,20.885,153.014
C06524=1092.475,294.396,417.751,177.389,20.888,153.014
C06525=1092.480,294.644,417.720,177.392,20.891,153.014
C06526=1092.486,294.892,417.690,177.395,20.894,153.014
C06527=1092.492,295.140,417.660,177.398,20.897,153.014
C06528=1092.498,295.388,417.630,177.401,20.899,153.014
C06529=1092.503,295.636,417.600,177.404,20.902,153.015
C06530=1092.509,295.884,417.570,177.407,20.905,153.015
C06531=1092.515,296.132,417.540,177.411,20.908,153.015
C06532=1092.521,296.380,417.509,177.414,20.911,153.015
C06533=1092.526,296.628,417.479,177.417,20.913,153.015
C06534=1092.532,296.877,417.448,177.420,20.916,153.015
C06535=1092.538,297.125,417.418,177.423,20.919,153.015
C06536=1092.543,297.373,417.388,177.426,20.922,153.016
C06537=1092.549,297.621,417.357,177.429,20.925,153.016
C06538=1092.555,297.869,417.328,177.432,20.927,153.016
C06539=1092.561,298.117,417.297,177.435,20.930,153.016
C06540=1092.566,298.365,417.266,177.438,20.933,153.016
C06541=1092.571,298.613,417.236,177.441,20.936,153.016
C06542=1092.577,298.861,417.206,177.444,20.939,153.017
C06543=1092.582,299.109,417.175,177.447,20.942,153.017
C06544=1092.588,299.357,417.144,177.450,20.945,153.017
C06545=1092.594,299.604,417.114,177.454,20.948,153.017
C06546=1092.599,299.853,417.083,177.457,20.951,153.017
C06547=1092.605,300.101,417.053,177.460,20.954,153.017
C06548=1092.610,300.349,417.022,177.463,20.957,153.017
C06549=1092.616,300.598,416.992,177.466,20.960,153.018
C06550=1092.622,300.845,416.961,177.469,20.963,153.018
C06551=1092.627,301.094,416.930,177.472,20.965,153.018
C06552=1092.633,301.341,416.900,177.475,20.968,153.018
C06553=1092.638,301.590,416.869,177.478,20.971,153.018
C06554=1092.644,301.837,416.838,177.481,20.974,153.019
C06555=1092.650,302.085,416.808,177.484,20.977,153.019
C06556=1092.655,302.333,416.777,177.487,20.980,153.019
C06557=1092.664,302.725,416.729,177.492,20.985,153.019
C06558=1092.673,303.116,416.680,177.497,20.989,153.019
C06559=1092.682,303.508,416.631,177.502,20.994,153.020
C06560=1092.691,303.900,416.582,177.507,20.999,153.020
C06561=1092.696,304.147,416.552,177.510,21.002,153.020
C06562=1092.702,304.396,416.521,177.513,21.005,153.020
C06563=1092.707,304.643,416.491,177.516,21.008,153.021
C06564=1092.713,304.892,416.459,177.519,21.011,153.021
C06565=1092.719,305.139,416.428,177.522,21.014,153.021
C06566=1092.724,305.388,416.397,177.525,21.017,153.021
C06567=1092.730,305.635,416.367,177.528,21.020,153.021
C06568=1092.736,305.884,416.335,177.531,21.023,153.021
C06569=1092.742,306.131,416.305,177.534,21.026,153.022
C06570=1092.747,306.380,416.274,177.537,21.029,153.022
C06571=1092.753,306.627,416.242,177.541,21.032,153.022
C06572=1092.759,306.876,416.211,177.544,21.035,153.022
C06573=1092.765,307.123,416.181,177.547,21.038,153.023
C06574=1092.770,307.371,416.149,177.550,21.041,153.023
C06575=1092.776,307.619,416.119,177.553,21.044,153.023
C06576=1092.782,307.867,416.087,177.556,21.047,153.023
C06577=1092.787,308.115,416.056,177.559,21.050,153.023
C06578=1092.793,308.363,416.025,177.562,21.053,153.023
C06579=1092.799,308.611,415.993,177.566,21.056,153.024
C06580=1092.804,308.859,415.963,177.569,21.059,153.024
C06581=1092.810,309.106,415.931,177.572,21.062,153.024
C06582=1092.816,309.355,415.901,177.575,21.065,153.024
C06583=1092.822,309.602,415.869,177.578,21.068,153.024
C06584=1092.827,309.851,415.838,177.581,21.071,153.025
C06585=1092.833,310.098,415.807,177.584,21.074,153.025
C06586=1092.839,310.347,415.776,177.588,21.078,153.025
C06587=1092.845,310.595,415.744,177.591,21.081,153.025
C06588=1092.851,310.842,415.713,177.594,21.084,153.025
C06589=1092.856,311.091,415.681,177.597,21.087,153.026
C06590=1092.862,311.338,415.650,177.600,21.090,153.026
C06591=1092.868,311.586,415.619,177.602,21.093,153.026
C06592=1092.873,311.834,415.587,177.606,21.096,153.026
C06593=1092.880,312.082,415.556,177.609,21.099,153.027
C06594=1092.885,312.330,415.525,177.612,21.102,153.027
C06595=1092.891,312.578,415.493,177.615,21.105,153.027
C06596=1092.897,312.826,415.462,177.618,21.108,153.027
C06597=1092.903,313.073,415.430,177.621,21.111,153.027
C06598=1092.908,313.322,415.399,177.624,21.114,153.028
C06599=1092.914,313.570,415.367,177.628,21.118,153.028
C06600=1092.921,313.818,415.336,177.631,21.121,153.028
C06601=1092.926,314.065,415.304,177.634,21.124,153.028
C06602=1092.932,314.314,415.273,177.637,21.127,153.029
C06603=1092.938,314.561,415.242,177.640,21.130,153.029
C06604=1092.944,314.809,415.210,177.644,21.133,153.029
C06605=1092.949,315.057,415.178,177.647,21.136,153.029
C06606=1092.955,315.305,415.146,177.649,21.140,153.029
C06607=1092.960,315.553,415.115,177.652,21.143,153.030
C06608=1092.966,315.801,415.083,177.655,21.146,153.030
C06609=1092.975,316.195,415.032,177.660,21.151,153.030
C06610=1092.984,316.590,414.982,177.665,21.157,153.031
C06611=1092.993,316.984,414.931,177.670,21.162,153.031
C06612=1093.002,317.379,414.881,177.675,21.167,153.032
C06613=1093.007,317.626,414.849,177.678,21.170,153.032
C06614=1093.013,317.874,414.817,177.681,21.173,153.032
C06615=1093.019,318.122,414.785,177.684,21.177,153.032
C06616=1093.025,318.370,414.753,177.687,21.180,153.033
C06617=1093.029,318.618,414.721,177.690,21.183,153.033
C06618=1093.035,318.866,414.689,177.693,21.187,153.033
C06619=1093.041,319.113,414.657,177.697,21.190,153.033
C06620=1093.047,319.361,414.625,177.700,21.194,153.034
C06621=1093.052,319.609,414.593,177.702,21.197,153.034
C06622=1093.058,319.857,414.561,177.705,21.200,153.034
C06623=1093.064,320.105,414.529,177.708,21.203,153.035
C06624=1093.069,320.353,414.497,177.712,21.207,153.035
C06625=1093.075,320.601,414.465,177.715,21.210,153.035
C06626=1093.080,320.849,414.433,177.718,21.213,153.035
C06627=1093.086,321.096,414.400,177.720,21.217,153.036
C06628=1093.092,321.344,414.369,177.724,21.221,153.036
C06629=1093.098,321.592,414.337,177.727,21.224,153.036
C06630=1093.103,321.841,414.304,177.730,21.227,153.037
C06631=1093.109,322.087,414.272,177.733,21.230,153.037
C06632=1093.115,322.336,414.240,177.737,21.234,153.037
C06633=1093.121,322.584,414.208,177.739,21.237,153.037
C06634=1093.126,322.831,414.176,177.742,21.240,153.038
C06635=1093.132,323.079,414.143,177.745,21.244,153.038
C06636=1093.138,323.327,414.111,177.749,21.247,153.038
C06637=1093.143,323.575,414.079,177.752,21.251,153.039
C06638=1093.149,323.823,414.046,177.755,21.254,153.039
C06639=1093.155,324.071,414.014,177.757,21.257,153.039
C06640=1093.160,324.319,413.982,177.761,21.261,153.040
C06641=1093.166,324.566,413.949,177.764,21.264,153.040
C06642=1093.172,324.814,413.917,177.767,21.268,153.040
C06643=1093.178,325.062,413.884,177.770,21.271,153.040
C06644=1093.183,325.310,413.852,177.773,21.275,153.041
C06645=1093.190,325.557,413.819,177.776,21.278,153.041
C06646=1093.195,325.806,413.787,177.779,21.281,153.042
C06647=1093.201,326.054,413.754,177.783,21.285,153.042
C06648=1093.206,326.301,413.722,177.786,21.288,153.042
C06649=1093.213,326.549,413.690,177.788,21.292,153.042
C06650=1093.218,326.797,413.657,177.792,21.296,153.043
C06651=1093.224,327.045,413.624,177.795,21.299,153.043
C06652=1093.230,327.292,413.593,177.798,21.302,153.043
C06653=1093.235,327.540,413.559,177.800,21.306,153.044
C06654=1093.241,327.788,413.527,177.804,21.309,153.044
C06655=1093.247,328.036,413.494,177.807,21.313,153.044
C06656=1093.253,328.284,413.461,177.810,21.316,153.045
C06657=1093.259,328.532,413.429,177.814,21.320,153.045
C06658=1093.264,328.779,413.396,177.816,21.323,153.045
C06659=1093.270,329.027,413.363,177.819,21.326,153.046
C06660=1093.276,329.275,413.331,177.823,21.330,153.046
C06661=1093.286,329.662,413.280,177.827,21.336,153.046
C06662=1093.295,330.050,413.229,177.832,21.341,153.047
C06663=1093.304,330.437,413.178,177.837,21.347,153.047
C06664=1093.313,330.824,413.126,177.842,21.352,153.048
C06665=1093.319,331.072,413.093,177.845,21.356,153.048
C06666=1093.325,331.320,413.060,177.848,21.359,153.049
C06667=1093.330,331.568,413.027,177.851,21.363,153.049
C06668=1093.336,331.816,412.995,177.854,21.366,153.049
C06669=1093.343,332.064,412.962,177.857,21.370,153.050
C06670=1093.348,332.311,412.929,177.861,21.374,153.050
C06671=1093.353,332.559,412.896,177.863,21.377,153.050
C06672=1093.360,332.806,412.863,177.867,21.381,153.051
C06673=1093.365,333.054,412.830,177.870,21.385,153.051
C06674=1093.371,333.302,412.796,177.872,21.388,153.052
C06675=1093.377,333.550,412.763,177.876,21.392,153.052
C06676=1093.383,333.798,412.730,177.879,21.396,153.052
C06677=1093.388,334.046,412.697,177.882,21.399,153.053
C06678=1093.394,334.293,412.663,177.885,21.403,153.053
C06679=1093.400,334.541,412.631,177.888,21.407,153.053
C06680=1093.405,334.788,412.598,177.891,21.411,153.054
C06681=1093.410,335.036,412.564,177.894,21.414,153.054
C06682=1093.417,335.284,412.532,177.897,21.418,153.055
C06683=1093.422,335.532,412.498,177.901,21.422,153.055
C06684=1093.428,335.780,412.465,177.903,21.426,153.055
C06685=1093.433,336.027,412.432,177.907,21.430,153.056
C06686=1093.440,336.275,412.399,177.909,21.433,153.056
C06687=1093.445,336.523,412.366,177.912,21.437,153.057
C06688=1093.451,336.771,412.332,177.916,21.441,153.057
C06689=1093.457,337.018,412.298,177.919,21.444,153.057
C06690=1093.463,337.266,412.265,177.922,21.449,153.058
C06691=1093.469,337.514,412.232,177.925,21.452,153.058
C06692=1093.474,337.762,412.199,177.928,21.456,153.059
C06693=1093.480,338.009,412.165,177.931,21.460,153.059
C06694=1093.485,338.257,412.131,177.934,21.464,153.059
C06695=1093.492,338.504,412.099,177.937,21.467,153.060
C06696=1093.497,338.752,412.065,177.940,21.471,153.060
C06697=1093.503,338.999,412.031,177.944,21.476,153.061
C06698=1093.509,339.247,411.998,177.946,21.479,153.061
C06699=1093.514,339.495,411.965,177.950,21.483,153.061
C06700=1093.520,339.743,411.931,177.952,21.487,153.062
C06701=1093.526,339.991,411.897,177.956,21.491,153.062
C06702=1093.532,340.239,411.863,177.959,21.495,153.063
C06703=1093.538,340.486,411.829,177.961,21.498,153.063
C06704=1093.543,340.734,411.796,177.965,21.503,153.064
C06705=1093.549,340.982,411.762,177.968,21.507,153.064
C06706=1093.555,341.229,411.729,177.971,21.510,153.064
C06707=1093.561,341.477,411.695,177.974,21.514,153.065
C06708=1093.566,341.725,411.661,177.977,21.519,153.065
C06709=1093.572,341.972,411.627,177.980,21.522,153.066
C06710=1093.578,342.220,411.594,177.983,21.527,153.066
C06711=1093.583,342.467,411.560,177.986,21.530,153.067
C06712=1093.589,342.715,411.527,177.990,21.534,153.067
C06713=1093.598,343.096,411.474,177.995,21.540,153.068
C06714=1093.607,343.478,411.422,177.999,21.547,153.069
C06715=1093.616,343.859,411.370,178.003,21.552,153.069
C06716=1093.625,344.241,411.318,178.008,21.559,153.070
C06717=1093.631,344.488,411.284,178.011,21.563,153.071
C06718=1093.637,344.737,411.250,178.014,21.567,153.071
C06719=1093.642,344.984,411.216,178.018,21.571,153.071
C06720=1093.648,345.231,411.182,178.020,21.575,153.072
C06721=1093.654,345.479,411.148,178.024,21.580,153.072
C06722=1093.660,345.727,411.114,178.027,21.584,153.073
C06723=1093.665,345.974,411.080,178.030,21.588,153.073
C06724=1093.671,346.222,411.045,178.033,21.592,153.074
C06725=1093.677,346.469,411.011,178.036,21.596,153.074
C06726=1093.683,346.717,410.978,178.039,21.600,153.075
C06727=1093.688,346.965,410.944,178.042,21.604,153.075
C06728=1093.694,347.212,410.910,178.045,21.609,153.076
C06729=1093.700,347.460,410.875,178.048,21.612,153.076
C06730=1093.706,347.708,410.841,178.051,21.617,153.077
C06731=1093.712,347.955,410.806,178.054,21.621,153.077
C06732=1093.717,348.202,410.772,178.057,21.625,153.078
C06733=1093.723,348.450,410.738,178.061,21.629,153.078
C06734=1093.729,348.698,410.703,178.063,21.634,153.079
C06735=1093.735,348.945,410.669,178.067,21.638,153.079
C06736=1093.740,349.193,410.635,178.069,21.642,153.080
C06737=1093.746,349.440,410.601,178.073,21.646,153.081
C06738=1093.752,349.688,410.566,178.075,21.650,153.081
C06739=1093.758,349.935,410.532,178.079,21.655,153.082
C06740=1093.763,350.183,410.497,178.082,21.659,153.082
C06741=1093.769,350.431,410.462,178.085,21.663,153.083
C06742=1093.775,350.678,410.428,178.088,21.668,153.083
C06743=1093.781,350.926,410.394,178.091,21.672,153.084
C06744=1093.786,351.173,410.360,178.094,21.676,153.084
C06745=1093.792,351.421,410.325,178.097,21.680,153.085
C06746=1093.798,351.668,410.291,178.100,21.685,153.085
C06747=1093.803,351.916,410.257,178.103,21.689,153.086
C06748=1093.810,352.163,410.221,178.106,21.693,153.086
C06749=1093.815,352.411,410.187,178.109,21.698,153.087
C06750=1093.821,352.658,410.153,178.112,21.702,153.088
C06751=1093.828,352.906,410.118,178.115,21.707,153.088
C06752=1093.833,353.154,410.084,178.119,21.711,153.089
C06753=1093.840,353.401,410.049,178.121,21.715,153.089
C06754=1093.845,353.649,410.014,178.124,21.720,153.090
C06755=1093.850,353.896,409.979,178.128,21.725,153.090
C06756=1093.857,354.144,409.944,178.130,21.728,153.091
C06757=1093.862,354.391,409.909,178.134,21.733,153.092
C06758=1093.868,354.639,409.875,178.137,21.738,153.092
C06759=1093.874,354.886,409.840,178.139,21.742,153.093
C06760=1093.879,355.134,409.806,178.143,21.747,153.093
C06761=1093.885,355.381,409.771,178.145,21.751,153.094
C06762=1093.891,355.629,409.735,178.148,21.756,153.095
C06763=1093.896,355.876,409.701,178.152,21.760,153.095
C06764=1093.903,356.124,409.665,178.154,21.764,153.096
C06765=1093.911,356.508,409.612,178.160,21.772,153.097
C06766=1093.921,356.892,409.558,178.164,21.779,153.098
C06767=1093.930,357.275,409.503,178.168,21.786,153.099
C06768=1093.938,357.660,409.449,178.173,21.792,153.099
C06769=1093.944,357.907,409.414,178.176,21.797,153.100
C06770=1093.951,358.154,409.379,178.180,21.802,153.101
C06771=1093.956,358.402,409.344,178.182,21.807,153.101
C06772=1093.962,358.649,409.308,178.185,21.811,153.102
C06773=1093.967,358.896,409.273,178.189,21.816,153.103
C06774=1093.974,359.144,409.239,178.192,21.821,153.103
C06775=1093.979,359.391,409.203,178.194,21.825,153.104
C06776=1093.985,359.639,409.168,178.198,21.830,153.104
C06777=1093.991,359.886,409.133,178.201,21.834,153.105
C06778=1093.997,360.134,409.098,178.203,21.839,153.106
C06779=1094.002,360.381,409.062,178.207,21.844,153.106
C06780=1094.008,360.629,409.027,178.210,21.848,153.107
C06781=1094.014,360.876,408.992,178.212,21.853,153.108
C06782=1094.020,361.123,408.957,178.216,21.858,153.108
C06783=1094.026,361.370,408.921,178.219,21.863,153.109
C06784=1094.032,361.618,408.886,178.222,21.868,153.110
C06785=1094.037,361.865,408.850,178.224,21.872,153.110
C06786=1094.043,362.113,408.815,178.228,21.877,153.111
C06787=1094.048,362.360,408.780,178.231,21.882,153.112
C06788=1094.054,362.608,408.744,178.234,21.887,153.112
C06789=1094.061,362.855,408.710,178.237,21.891,153.113
C06790=1094.067,363.102,408.674,178.240,21.896,153.114
C06791=1094.073,363.350,408.638,178.243,21.901,153.114
C06792=1094.078,363.597,408.603,178.246,21.906,153.115
C06793=1094.084,363.845,408.567,178.248,21.911,153.116
C06794=1094.090,364.092,408.532,178.252,21.916,153.117
C06795=1094.096,364.339,408.496,178.255,21.921,153.117
C06796=1094.102,364.587,408.460,178.258,21.926,153.118
C06797=1094.107,364.834,408.425,178.260,21.930,153.119
C06798=1094.113,365.082,408.389,178.264,21.935,153.119
C06799=1094.119,365.329,408.354,178.267,21.940,153.120
C06800=1094.125,365.576,408.318,178.270,21.945,153.121
C06801=1094.131,365.823,408.282,178.273,21.950,153.122
C06802=1094.136,366.070,408.246,178.275,21.955,153.122
C06803=1094.142,366.318,408.210,178.279,21.960,153.123
C06804=1094.148,366.566,408.175,178.282,21.965,153.124
C06805=1094.154,366.813,408.139,178.285,21.970,153.125
C06806=1094.160,367.060,408.104,178.288,21.975,153.125
C06807=1094.166,367.307,408.068,178.290,21.980,153.126
C06808=1094.171,367.555,408.031,178.293,21.985,153.127
C06809=1094.177,367.802,407.995,178.297,21.990,153.128
C06810=1094.183,368.049,407.959,178.300,21.996,153.128
C06811=1094.189,368.296,407.924,178.303,22.001,153.129
C06812=1094.195,368.544,407.888,178.305,22.006,153.130
C06813=1094.200,368.790,407.852,178.308,22.011,153.131
C06814=1094.206,369.038,407.816,178.311,22.016,153.131
C06815=1094.212,369.286,407.780,178.314,22.021,153.132
C06816=1094.218,369.533,407.743,178.318,22.026,153.133
C06817=1094.227,369.932,407.685,178.323,22.035,153.134
C06818=1094.237,370.331,407.627,178.326,22.043,153.136
C06819=1094.246,370.731,407.569,178.331,22.051,153.137
C06820=1094.255,371.130,407.511,178.336,22.060,153.138
C06821=1094.262,371.377,407.474,178.340,22.065,153.139
C06822=1094.267,371.624,407.439,178.342,22.071,153.140
C06823=1094.273,371.871,407.402,178.346,22.076,153.140
C06824=1094.279,372.119,407.366,178.349,22.081,153.141
C06825=1094.285,372.366,407.330,178.351,22.086,153.142
C06826=1094.291,372.613,407.293,178.354,22.091,153.143
C06827=1094.296,372.860,407.257,178.357,22.097,153.144
C06828=1094.302,373.107,407.221,178.360,22.102,153.145
C06829=1094.309,373.354,407.184,178.363,22.107,153.145
C06830=1094.314,373.602,407.148,178.366,22.113,153.146
C06831=1094.320,373.849,407.112,178.369,22.118,153.147
C06832=1094.327,374.096,407.075,178.372,22.124,153.148
C06833=1094.331,374.344,407.039,178.375,22.129,153.149
C06834=1094.338,374.591,407.003,178.378,22.135,153.150
C06835=1094.343,374.838,406.966,178.380,22.140,153.151
C06836=1094.350,375.085,406.929,178.383,22.145,153.151
C06837=1094.355,375.333,406.892,178.386,22.151,153.152
C06838=1094.361,375.579,406.856,178.389,22.156,153.153
C06839=1094.366,375.827,406.820,178.392,22.162,153.154
C06840=1094.373,376.074,406.783,178.395,22.167,153.155
C06841=1094.378,376.321,406.746,178.398,22.173,153.156
C06842=1094.385,376.568,406.710,178.401,22.179,153.157
C06843=1094.390,376.816,406.673,178.404,22.184,153.158
C06844=1094.396,377.063,406.636,178.407,22.190,153.158
C06845=1094.401,377.309,406.600,178.410,22.195,153.159
C06846=1094.408,377.556,406.563,178.413,22.201,153.160
C06847=1094.413,377.804,406.526,178.416,22.207,153.161
C06848=1094.419,378.051,406.489,178.419,22.212,153.162
C06849=1094.425,378.298,406.453,178.422,22.218,153.163
C06850=1094.431,378.546,406.416,178.425,22.224,153.164
C06851=1094.437,378.793,406.379,178.428,22.229,153.165
C06852=1094.443,379.040,406.342,178.431,22.235,153.166
C06853=1094.449,379.287,406.306,178.434,22.241,153.167
C06854=1094.455,379.534,406.269,178.437,22.246,153.168
C06855=1094.461,379.781,406.231,178.439,22.252,153.169
C06856=1094.467,380.028,406.195,178.442,22.258,153.170
C06857=1094.472,380.275,406.158,178.445,22.263,153.170
C06858=1094.478,380.522,406.121,178.448,22.269,153.171
C06859=1094.484,380.769,406.084,178.451,22.275,153.172
C06860=1094.490,381.016,406.047,178.454,22.281,153.173
C06861=1094.496,381.263,406.010,178.457,22.287,153.174
C06862=1094.502,381.510,405.973,178.460,22.293,153.175
C06863=1094.507,381.758,405.936,178.463,22.299,153.176
C06864=1094.514,382.005,405.898,178.466,22.304,153.177
C06865=1094.520,382.252,405.862,178.469,22.310,153.178
C06866=1094.526,382.500,405.825,178.471,22.316,153.179
C06867=1094.532,382.746,405.787,178.474,22.322,153.180
C06868=1094.537,382.994,405.750,178.477,22.328,153.181
C06869=1094.543,383.206,405.718,178.480,22.333,153.182
C06870=1094.548,383.420,405.685,178.482,22.338,153.183
C06871=1094.552,383.633,405.654,178.484,22.343,153.184
C06872=1094.557,383.847,405.621,178.487,22.349,153.185
C06873=1094.563,384.060,405.589,178.490,22.354,153.186
C06874=1094.568,384.272,405.557,178.492,22.359,153.186
C06875=1094.573,384.486,405.524,178.495,22.364,153.187
C06876=1094.578,384.700,405.492,178.497,22.370,153.188
C06877=1094.584,384.947,405.455,178.500,22.376,153.189
C06878=1094.589,385.194,405.417,178.503,22.381,153.190
C06879=1094.595,385.441,405.380,178.506,22.388,153.191
C06880=1094.602,385.687,405.343,178.509,22.394,153.192
C06881=1094.607,385.935,405.306,178.512,22.400,153.193
C06882=1094.613,386.181,405.268,178.515,22.406,153.194
C06883=1094.619,386.429,405.231,178.517,22.413,153.196
C06884=1094.625,386.676,405.193,178.520,22.419,153.197
C06885=1094.631,386.922,405.155,178.523,22.425,153.198
C06886=1094.637,387.169,405.117,178.526,22.431,153.199
C06887=1094.642,387.416,405.080,178.529,22.438,153.200
C06888=1094.649,387.664,405.042,178.532,22.444,153.201
C06889=1094.655,387.911,405.005,178.535,22.450,153.202
C06890=1094.661,388.157,404.967,178.537,22.456,153.203
C06891=1094.666,388.405,404.930,178.540,22.463,153.204
C06892=1094.672,388.651,404.892,178.543,22.469,153.205
C06893=1094.678,388.898,404.854,178.546,22.476,153.207
C06894=1094.684,389.146,404.816,178.549,22.482,153.208
C06895=1094.690,389.392,404.778,178.552,22.488,153.209
C06896=1094.696,389.639,404.741,178.555,22.494,153.210
C06897=1094.702,389.886,404.703,178.557,22.501,153.211
C06898=1094.708,390.133,404.665,178.560,22.507,153.212
C06899=1094.714,390.381,404.628,178.564,22.514,153.213
C06900=1094.719,390.628,404.589,178.566,22.520,153.214
C06901=1094.725,390.874,404.552,178.569,22.527,153.216
C06902=1094.731,391.121,404.514,178.572,22.533,153.217
C06903=1094.738,391.369,404.476,178.575,22.540,153.218
C06904=1094.744,391.615,404.438,178.578,22.546,153.219
C06905=1094.750,391.861,404.399,178.581,22.553,153.220
C06906=1094.756,392.109,404.361,178.583,22.559,153.221
C06907=1094.762,392.356,404.324,178.586,22.565,153.222
C06908=1094.767,392.603,404.285,178.589,22.573,153.224
C06909=1094.774,392.850,404.247,178.592,22.579,153.225
C06910=1094.780,393.097,404.209,178.595,22.586,153.226
C06911=1094.786,393.344,404.172,178.597,22.592,153.227
C06912=1094.792,393.591,404.133,178.601,22.599,153.228
C06913=1094.798,393.838,404.094,178.603,22.606,153.230
C06914=1094.804,394.084,404.057,178.606,22.612,153.231
C06915=1094.809,394.332,404.018,178.608,22.619,153.232
C06916=1094.815,394.579,403.980,178.612,22.626,153.233
C06917=1094.822,394.825,403.942,178.614,22.633,153.235
C06918=1094.827,395.073,403.903,178.617,22.640,153.236
C06919=1094.833,395.319,403.865,178.620,22.646,153.237
C06920=1094.838,395.566,403.827,178.623,22.654,153.238
C06921=1094.845,395.813,403.788,178.626,22.660,153.240
C06922=1094.851,396.060,403.750,178.628,22.667,153.241
C06923=1094.857,396.307,403.711,178.631,22.674,153.242
C06924=1094.863,396.554,403.673,178.634,22.681,153.244
C06925=1094.868,396.774,403.639,178.637,22.688,153.245
C06926=1094.873,396.993,403.604,178.639,22.693,153.246
C06927=1094.878,397.213,403.570,178.641,22.700,153.247
C06928=1094.883,397.433,403.536,178.644,22.706,153.248
C06929=1094.889,397.653,403.501,178.647,22.712,153.249
C06930=1094.895,397.872,403.467,178.649,22.718,153.250
C06931=1094.900,398.092,403.433,178.651,22.725,153.252
C06932=1094.905,398.312,403.399,178.654,22.731,153.253
C06933=1094.911,398.559,403.360,178.656,22.738,153.254
C06934=1094.918,398.805,403.321,178.660,22.745,153.255
C06935=1094.923,399.053,403.282,178.662,22.753,153.257
C06936=1094.929,399.299,403.244,178.665,22.760,153.258
C06937=1094.935,399.547,403.205,178.668,22.767,153.259
C06938=1094.941,399.793,403.166,178.670,22.774,153.261
C06939=1094.948,400.040,403.127,178.673,22.781,153.262
C06940=1094.953,400.287,403.089,178.676,22.789,153.264
C06941=1094.959,400.534,403.049,178.679,22.796,153.265
C06942=1094.965,400.780,403.011,178.682,22.804,153.266
C06943=1094.971,401.027,402.972,178.684,22.810,153.268
C06944=1094.976,401.275,402.933,178.688,22.818,153.269
C06945=1094.983,401.521,402.894,178.690,22.825,153.270
C06946=1094.989,401.768,402.855,178.692,22.833,153.272
C06947=1094.995,402.015,402.816,178.696,22.840,153.273
C06948=1095.001,402.262,402.777,178.698,22.848,153.275
C06949=1095.007,402.509,402.739,178.701,22.855,153.276
C06950=1095.013,402.756,402.699,178.704,22.863,153.278
C06951=1095.018,403.002,402.660,178.707,22.870,153.279
C06952=1095.025,403.249,402.621,178.709,22.877,153.280
C06953=1095.031,403.496,402.582,178.713,22.885,153.282
C06954=1095.036,403.743,402.543,178.715,22.892,153.283
C06955=1095.043,403.990,402.503,178.718,22.901,153.285
C06956=1095.049,404.237,402.464,178.720,22.908,153.286
C06957=1095.055,404.483,402.426,178.724,22.916,153.288
C06958=1095.061,404.730,402.386,178.726,22.923,153.289
C06959=1095.067,404.977,402.347,178.729,22.931,153.291
C06960=1095.072,405.224,402.308,178.731,22.939,153.292
C06961=1095.079,405.471,402.268,178.735,22.946,153.294
C06962=1095.085,405.718,402.229,178.737,22.954,153.295
C06963=1095.091,405.965,402.189,178.740,22.962,153.297
C06964=1095.096,406.211,402.150,178.743,22.970,153.298
C06965=1095.103,406.458,402.110,178.745,22.977,153.300
C06966=1095.109,406.705,402.071,178.749,22.986,153.301
C06967=1095.114,406.952,402.032,178.751,22.993,153.303
C06968=1095.120,407.198,401.991,178.754,23.001,153.304
C06969=1095.127,407.445,401.952,178.756,23.009,153.306
C06970=1095.133,407.693,401.913,178.759,23.017,153.307
C06971=1095.138,407.939,401.874,178.762,23.025,153.309
C06972=1095.144,408.186,401.833,178.764,23.033,153.311
C06973=1095.151,408.433,401.794,178.768,23.042,153.312
C06974=1095.157,408.679,401.754,178.771,23.050,153.314
C06975=1095.162,408.926,401.715,178.773,23.058,153.315
C06976=1095.168,409.173,401.675,178.776,23.066,153.317
C06977=1095.175,409.419,401.635,178.779,23.074,153.319
C06978=1095.180,409.667,401.595,178.781,23.082,153.320
C06979=1095.186,409.913,401.555,178.784,23.091,153.322
C06980=1095.192,410.160,401.516,178.787,23.099,153.323
C06981=1095.198,410.380,401.481,178.790,23.106,153.325
C06982=1095.203,410.600,401.445,178.792,23.114,153.326
C06983=1095.208,410.820,401.409,178.794,23.121,153.328
C06984=1095.214,411.040,401.374,178.797,23.128,153.329
C06985=1095.219,411.260,401.339,178.799,23.136,153.331
C06986=1095.224,411.480,401.303,178.801,23.143,153.332
C06987=1095.230,411.699,401.267,178.804,23.150,153.334
C06988=1095.235,411.919,401.231,178.806,23.158,153.335
C06989=1095.242,412.167,401.192,178.809,23.167,153.337
C06990=1095.247,412.413,401.151,178.812,23.175,153.339
C06991=1095.254,412.660,401.111,178.815,23.184,153.340
C06992=1095.260,412.907,401.071,178.818,23.192,153.342
C06993=1095.266,413.154,401.031,178.820,23.201,153.344
C06994=1095.271,413.400,400.991,178.823,23.209,153.346
C06995=1095.277,413.646,400.951,178.826,23.218,153.347
C06996=1095.284,413.893,400.910,178.829,23.227,153.349
C06997=1095.290,414.139,400.870,178.832,23.235,153.351
C06998=1095.296,414.387,400.830,178.834,23.244,153.353
C06999=1095.302,414.633,400.790,178.837,23.252,153.354
C07000=1095.308,414.880,400.750,178.840,23.261,153.356
C07001=1095.314,415.126,400.709,178.843,23.270,153.358
C07002=1095.320,415.373,400.669,178.846,23.279,153.360
C07003=1095.327,415.619,400.629,178.848,23.288,153.361
C07004=1095.332,415.866,400.588,178.851,23.297,153.363
C07005=1095.339,416.113,400.548,178.853,23.305,153.365
C07006=1095.346,416.360,400.508,178.856,23.314,153.367
C07007=1095.351,416.607,400.467,178.859,23.323,153.369
C07008=1095.358,416.853,400.427,178.862,23.332,153.370
C07009=1095.363,417.100,400.386,178.865,23.341,153.372
C07010=1095.370,417.347,400.346,178.867,23.350,153.374
C07011=1095.376,417.593,400.304,178.870,23.359,153.376
C07012=1095.382,417.839,400.264,178.873,23.369,153.378
C07013=1095.388,418.086,400.223,178.876,23.378,153.380
C07014=1095.393,418.333,400.183,178.878,23.387,153.382
C07015=1095.400,418.580,400.142,178.881,23.396,153.384
C07016=1095.406,418.826,400.101,178.884,23.405,153.386
C07017=1095.412,419.072,400.061,178.887,23.415,153.387
C07018=1095.418,419.319,400.020,178.890,23.424,153.389
C07019=1095.424,419.565,399.979,178.892,23.433,153.391
C07020=1095.430,419.812,399.939,178.895,23.443,153.393
C07021=1095.436,420.059,399.898,178.898,23.452,153.395
C07022=1095.442,420.305,399.857,178.901,23.461,153.397
C07023=1095.449,420.552,399.816,178.903,23.471,153.399
C07024=1095.455,420.798,399.774,178.906,23.480,153.401
C07025=1095.461,421.045,399.734,178.909,23.490,153.403
C07026=1095.467,421.291,399.693,178.911,23.499,153.405
C07027=1095.473,421.538,399.652,178.914,23.509,153.407
C07028=1095.479,421.784,399.611,178.917,23.518,153.409
C07029=1095.485,422.031,399.570,178.919,23.528,153.411
C07030=1095.491,422.277,399.529,178.922,23.538,153.413
C07031=1095.498,422.523,399.488,178.925,23.547,153.415
C07032=1095.504,422.770,399.447,178.928,23.557,153.417
C07033=1095.510,423.016,399.406,178.931,23.567,153.419
C07034=1095.516,423.264,399.364,178.934,23.577,153.421
C07035=1095.522,423.510,399.323,178.936,23.587,153.423
C07036=1095.528,423.756,399.282,178.939,23.596,153.425
C07037=1095.533,423.984,399.244,178.942,23.606,153.427
C07038=1095.539,424.210,399.206,178.943,23.615,153.429
C07039=1095.545,424.438,399.168,178.946,23.624,153.431
C07040=1095.551,424.665,399.130,178.949,23.633,153.433
C07041=1095.556,424.892,399.091,178.952,23.643,153.435
C07042=1095.562,425.119,399.053,178.954,23.651,153.437
C07043=1095.568,425.346,399.015,178.957,23.661,153.439
C07044=1095.573,425.573,398.976,178.959,23.671,153.441
C07045=1095.579,425.819,398.936,178.962,23.680,153.443
C07046=1095.586,426.066,398.894,178.964,23.691,153.445
C07047=1095.592,426.312,398.852,178.967,23.701,153.447
C07048=1095.598,426.558,398.811,178.970,23.711,153.450
C07049=1095.604,426.805,398.769,178.973,23.722,153.452
C07050=1095.610,427.052,398.727,178.975,23.732,153.454
C07051=1095.616,427.298,398.686,178.978,23.742,153.456
C07052=1095.623,427.545,398.644,178.981,23.753,153.458
C07053=1095.629,427.791,398.603,178.983,23.763,153.461
C07054=1095.635,428.037,398.561,178.986,23.773,153.463
C07055=1095.641,428.284,398.519,178.988,23.784,153.465
C07056=1095.648,428.530,398.477,178.992,23.794,153.467
C07057=1095.654,428.777,398.435,178.994,23.804,153.470
C07058=1095.660,429.023,398.394,178.997,23.815,153.472
C07059=1095.666,429.269,398.353,179.000,23.826,153.474
C07060=1095.672,429.516,398.309,179.002,23.837,153.477
C07061=1095.678,429.762,398.268,179.005,23.847,153.479
C07062=1095.685,430.009,398.226,179.008,23.858,153.481
C07063=1095.691,430.254,398.184,179.010,23.869,153.484
C07064=1095.697,430.500,398.143,179.014,23.880,153.486
C07065=1095.703,430.747,398.099,179.016,23.891,153.488
C07066=1095.709,430.993,398.058,179.018,23.901,153.490
C07067=1095.715,431.240,398.016,179.021,23.913,153.493
C07068=1095.722,431.486,397.974,179.024,23.924,153.495
C07069=1095.728,431.733,397.932,179.027,23.935,153.498
C07070=1095.734,431.978,397.889,179.029,23.946,153.500
C07071=1095.741,432.225,397.847,179.032,23.957,153.503
C07072=1095.747,432.471,397.805,179.035,23.968,153.505
C07073=1095.753,432.717,397.763,179.037,23.979,153.507
C07074=1095.759,432.964,397.721,179.040,23.990,153.510
C07075=1095.765,433.210,397.678,179.043,24.001,153.512
C07076=1095.772,433.456,397.636,179.046,24.013,153.515
C07077=1095.778,433.702,397.593,179.048,24.024,153.517
C07078=1095.784,433.948,397.551,179.051,24.036,153.520
C07079=1095.790,434.195,397.508,179.053,24.047,153.522
C07080=1095.796,434.441,397.466,179.056,24.059,153.525
C07081=1095.802,434.687,397.423,179.059,24.070,153.527
C07082=1095.809,434.933,397.381,179.062,24.082,153.530
C07083=1095.815,435.179,397.338,179.064,24.093,153.532
C07084=1095.821,435.426,397.296,179.067,24.105,153.535
C07085=1095.827,435.672,397.253,179.069,24.117,153.538
C07086=1095.833,435.918,397.211,179.072,24.129,153.540
C07087=1095.839,436.164,397.168,179.075,24.141,153.543
C07088=1095.846,436.411,397.125,179.077,24.152,153.545
C07089=1095.851,436.657,397.082,179.080,24.164,153.548
C07090=1095.858,436.903,397.040,179.082,24.176,153.551
C07091=1095.865,437.149,396.996,179.086,24.188,153.553
C07092=1095.871,437.394,396.954,179.088,24.200,153.556
C07093=1095.877,437.648,396.910,179.090,24.212,153.559
C07094=1095.884,437.901,396.866,179.093,24.225,153.562
C07095=1095.891,438.154,396.822,179.096,24.237,153.564
C07096=1095.897,438.407,396.777,179.099,24.250,153.567
C07097=1095.904,438.653,396.734,179.101,24.261,153.570
C07098=1095.909,438.899,396.692,179.104,24.274,153.573
C07099=1095.916,439.145,396.649,179.107,24.286,153.575
C07100=1095.922,439.391,396.605,179.110,24.298,153.578
C07101=1095.929,439.639,396.562,179.112,24.311,153.581
C07102=1095.935,439.886,396.519,179.115,24.323,153.583
C07103=1095.941,440.134,396.475,179.118,24.336,153.586
C07104=1095.948,440.381,396.432,179.121,24.348,153.589
C07105=1095.954,440.627,396.389,179.123,24.361,153.592
C07106=1095.960,440.873,396.346,179.125,24.373,153.595
C07107=1095.966,441.119,396.303,179.128,24.386,153.598
C07108=1095.973,441.365,396.259,179.131,24.399,153.601
C07109=1095.979,441.612,396.216,179.133,24.411,153.603
C07110=1095.986,441.857,396.172,179.136,24.424,153.606
C07111=1095.992,442.103,396.129,179.139,24.437,153.609
C07112=1095.998,442.349,396.086,179.142,24.450,153.612
C07113=1096.004,442.595,396.042,179.143,24.463,153.615
C07114=1096.011,442.841,395.998,179.146,24.476,153.618
C07115=1096.017,443.087,395.954,179.149,24.489,153.621
C07116=1096.023,443.334,395.911,179.152,24.502,153.624
C07117=1096.029,443.579,395.868,179.154,24.515,153.627
C07118=1096.036,443.825,395.824,179.157,24.529,153.630
C07119=1096.042,444.071,395.780,179.159,24.541,153.633
C07120=1096.048,444.317,395.736,179.162,24.555,153.636
C07121=1096.056,444.563,395.693,179.163,24.568,153.639
C07122=1096.062,444.809,395.650,179.166,24.581,153.642
C07123=1096.068,445.055,395.606,179.168,24.594,153.645
C07124=1096.075,445.301,395.562,179.170,24.608,153.648
C07125=1096.081,445.547,395.518,179.170,24.621,153.652
C07126=1096.087,445.793,395.474,179.172,24.634,153.655
C07127=1096.093,446.039,395.430,179.173,24.647,153.658
C07128=1096.100,446.285,395.386,179.174,24.660,153.661
C07129=1096.106,446.531,395.342,179.175,24.673,153.664
C07130=1096.113,446.777,395.298,179.175,24.686,153.667
C07131=1096.119,447.023,395.254,179.176,24.699,153.671
C07132=1096.126,447.269,395.210,179.177,24.712,153.674
C07133=1096.132,447.515,395.166,179.177,24.725,153.677
C07134=1096.138,447.761,395.122,179.177,24.738,153.680
C07135=1096.144,448.007,395.078,179.177,24.751,153.684
C07136=1096.151,448.253,395.034,179.177,24.764,153.687
C07137=1096.157,448.498,394.989,179.177,24.777,153.690
C07138=1096.164,448.744,394.945,179.177,24.790,153.694
C07139=1096.169,448.990,394.901,179.175,24.803,153.697
C07140=1096.176,449.236,394.857,179.175,24.816,153.701
C07141=1096.183,449.482,394.813,179.174,24.829,153.704
C07142=1096.189,449.728,394.769,179.174,24.842,153.707
C07143=1096.196,449.973,394.724,179.173,24.855,153.711
C07144=1096.203,450.219,394.681,179.172,24.867,153.714
C07145=1095.812,450.212,394.516,179.116,25.079,153.774
C07146=1095.804,449.965,394.560,179.117,25.067,153.771
C07147=1095.797,449.719,394.604,179.118,25.054,153.768
C07148=1095.791,449.474,394.648,179.118,25.040,153.765
C07149=1095.785,449.228,394.693,179.119,25.028,153.761
C07150=1095.778,448.982,394.737,179.119,25.015,153.758
C07151=1095.772,448.736,394.781,179.120,25.002,153.754
C07152=1095.765,448.490,394.825,179.120,24.989,153.751
C07153=1095.758,448.244,394.870,179.120,24.976,153.748
C07154=1095.752,447.998,394.914,179.120,24.962,153.744
C07155=1095.746,447.752,394.958,179.120,24.950,153.741
C07156=1095.740,447.506,395.002,179.120,24.936,153.738
C07157=1095.733,447.261,395.047,179.120,24.923,153.735
C07158=1095.726,447.015,395.090,179.119,24.910,153.731
C07159=1095.721,446.768,395.135,179.119,24.897,153.728
C07160=1095.714,446.522,395.179,179.118,24.884,153.725
C07161=1095.708,446.276,395.223,179.117,24.871,153.722
C07162=1095.701,446.031,395.266,179.115,24.857,153.718
C07163=1095.695,445.785,395.310,179.115,24.844,153.715
C07164=1095.688,445.539,395.355,179.113,24.831,153.712
C07165=1095.682,445.293,395.399,179.112,24.818,153.709
C07166=1095.675,445.047,395.442,179.110,24.805,153.706
C07167=1095.669,444.801,395.486,179.108,24.792,153.703
C07168=1095.663,444.555,395.530,179.105,24.778,153.700
C07169=1095.656,444.309,395.574,179.103,24.765,153.697
C07170=1095.650,444.063,395.618,179.101,24.752,153.693
C07171=1095.644,443.817,395.661,179.099,24.738,153.690
C07172=1095.637,443.571,395.705,179.096,24.725,153.687
C07173=1095.631,443.325,395.749,179.093,24.712,153.684
C07174=1095.625,443.080,395.792,179.090,24.699,153.681
C07175=1095.619,442.834,395.836,179.087,24.686,153.678
C07176=1095.612,442.588,395.880,179.086,24.673,153.676
C07177=1095.606,442.341,395.923,179.083,24.660,153.673
C07178=1095.600,442.095,395.967,179.080,24.647,153.670
C07179=1095.592,441.849,396.010,179.077,24.634,153.667
C07180=1095.586,441.603,396.054,179.074,24.621,153.664
C07181=1095.580,441.357,396.097,179.072,24.608,153.661
C07182=1095.574,441.112,396.141,179.069,24.595,153.658
C07183=1095.568,440.865,396.184,179.066,24.582,153.655
C07184=1095.562,440.619,396.228,179.063,24.570,153.652
C07185=1095.554,440.373,396.271,179.061,24.557,153.649
C07186=1095.549,440.127,396.314,179.058,24.545,153.647
C07187=1095.543,439.881,396.357,179.055,24.532,153.644
C07188=1095.536,439.635,396.400,179.052,24.520,153.641
C07189=1095.529,439.389,396.443,179.050,24.507,153.638
C07190=1095.523,439.144,396.486,179.047,24.495,153.636
C07191=1095.517,438.898,396.529,179.044,24.482,153.633
C07192=1095.510,438.652,396.572,179.042,24.471,153.630
C07193=1095.504,438.407,396.615,179.039,24.458,153.627
C07194=1095.498,438.162,396.658,179.037,24.446,153.625
C07195=1095.491,437.917,396.701,179.034,24.434,153.622
C07196=1095.485,437.671,396.743,179.031,24.422,153.619
C07197=1095.478,437.426,396.786,179.028,24.410,153.617
C07198=1095.472,437.180,396.829,179.025,24.398,153.614
C07199=1095.466,436.934,396.872,179.023,24.386,153.611
C07200=1095.460,436.688,396.915,179.020,24.374,153.609
C07201=1095.453,436.443,396.958,179.017,24.362,153.606
C07202=1095.447,436.196,397.001,179.015,24.350,153.603
C07203=1095.441,435.949,397.044,179.012,24.338,153.601
C07204=1095.435,435.704,397.086,179.010,24.326,153.598
C07205=1095.429,435.457,397.129,179.006,24.315,153.595
C07206=1095.422,435.211,397.172,179.004,24.303,153.593
C07207=1095.416,434.965,397.215,179.001,24.291,153.590
C07208=1095.410,434.719,397.257,178.999,24.280,153.588
C07209=1095.404,434.472,397.299,178.996,24.268,153.585
C07210=1095.397,434.226,397.342,178.992,24.256,153.583
C07211=1095.392,433.980,397.384,178.990,24.245,153.580
C07212=1095.385,433.734,397.427,178.987,24.233,153.578
C07213=1095.379,433.488,397.469,178.985,24.222,153.575
C07214=1095.373,433.242,397.512,178.982,24.211,153.573
C07215=1095.367,432.995,397.554,178.979,24.199,153.570
C07216=1095.361,432.749,397.597,178.977,24.188,153.568
C07217=1095.354,432.503,397.639,178.974,24.177,153.565
C07218=1095.348,432.256,397.681,178.971,24.166,153.563
C07219=1095.341,432.010,397.723,178.968,24.154,153.560
C07220=1095.335,431.764,397.766,178.966,24.143,153.558
C07221=1095.329,431.517,397.808,178.962,24.132,153.556
C07222=1095.323,431.272,397.850,178.960,24.121,153.553
C07223=1095.316,431.025,397.892,178.958,24.110,153.551
C07224=1095.311,430.779,397.935,178.954,24.099,153.548
C07225=1095.305,430.533,397.976,178.952,24.088,153.546
C07226=1095.298,430.286,398.019,178.949,24.077,153.544
C07227=1095.292,430.040,398.060,178.946,24.066,153.541
C07228=1095.285,429.794,398.103,178.944,24.056,153.539
C07229=1095.280,429.547,398.145,178.940,24.045,153.537
C07230=1095.273,429.301,398.187,178.938,24.034,153.534
C07231=1095.267,429.055,398.229,178.935,24.023,153.532
C07232=1095.261,428.809,398.270,178.933,24.013,153.530
C07233=1095.254,428.562,398.312,178.929,24.002,153.527
C07234=1095.248,428.316,398.354,178.927,23.992,153.525
C07235=1095.242,428.069,398.396,178.924,23.981,153.523
C07236=1095.236,427.823,398.438,178.921,23.970,153.521
C07237=1095.229,427.576,398.479,178.919,23.960,153.518
C07238=1095.223,427.330,398.521,178.916,23.950,153.516
C07239=1095.217,427.084,398.562,178.913,23.939,153.514
C07240=1095.210,426.838,398.605,178.910,23.929,153.512
C07241=1095.204,426.591,398.646,178.907,23.919,153.510
C07242=1095.199,426.345,398.688,178.905,23.908,153.507
C07243=1095.192,426.098,398.730,178.902,23.898,153.505
C07244=1095.186,425.852,398.771,178.899,23.888,153.503
C07245=1095.180,425.606,398.813,178.896,23.877,153.501
C07246=1095.174,425.378,398.851,178.893,23.868,153.499
C07247=1095.169,425.151,398.889,178.891,23.859,153.497
C07248=1095.162,424.923,398.927,178.889,23.849,153.495
C07249=1095.157,424.695,398.966,178.886,23.840,153.493
C07250=1095.152,424.468,399.004,178.884,23.831,153.491
C07251=1095.146,424.240,399.043,178.881,23.821,153.489
C07252=1095.140,424.013,399.080,178.878,23.812,153.487
C07253=1095.135,423.785,399.118,178.876,23.803,153.485
C07254=1095.128,423.538,399.160,178.873,23.793,153.483
C07255=1095.122,423.292,399.201,178.870,23.783,153.481
C07256=1095.116,423.046,399.243,178.867,23.773,153.479
C07257=1095.111,422.799,399.283,178.865,23.763,153.477
C07258=1095.104,422.552,399.325,178.862,23.753,153.475
C07259=1095.097,422.306,399.366,178.859,23.744,153.473
C07260=1095.092,422.059,399.407,178.857,23.734,153.471
C07261=1095.086,421.813,399.448,178.854,23.725,153.469
C07262=1095.079,421.567,399.490,178.851,23.715,153.467
C07263=1095.073,421.320,399.530,178.847,23.705,153.465
C07264=1095.067,421.074,399.572,178.845,23.696,153.463
C07265=1095.061,420.827,399.612,178.842,23.686,153.461
C07266=1095.055,420.581,399.653,178.839,23.676,153.459
C07267=1095.049,420.334,399.694,178.836,23.667,153.457
C07268=1095.042,420.087,399.735,178.834,23.657,153.455
C07269=1095.036,419.841,399.776,178.831,23.648,153.453
C07270=1095.030,419.594,399.817,178.828,23.639,153.451
C07271=1095.024,419.348,399.858,178.825,23.629,153.449
C07272=1095.018,419.101,399.898,178.823,23.620,153.447
C07273=1095.011,418.855,399.939,178.820,23.611,153.445
C07274=1095.006,418.608,399.980,178.817,23.601,153.443
C07275=1095.000,418.362,400.021,178.814,23.592,153.441
C07276=1094.993,418.116,400.062,178.811,23.583,153.439
C07277=1094.987,417.868,400.103,178.808,23.573,153.437
C07278=1094.982,417.653,400.138,178.806,23.565,153.436
C07279=1094.976,417.437,400.173,178.804,23.558,153.434
